Omron CX-Programmer project NewProject (CX-Programmer 9.61)

# PLC NewPLC1: CJ2M CPU35
I/O table (CPU CJ2M-CPU35): rack 0 slot 0 CJ1W-ID211; rack 0 slot 1 CJ1W-ID211; rack 0 slot 2 CJ1W-ID211; rack 0 slot 3 CJ1W-ID211; rack 0 slot 4 CJ1W-ID211; rack 0 slot 5 CJ1W-OD211; rack 0 slot 6 CJ1W-OD211; rack 0 slot 7 CJ1W-OD211; rack 0 slot 11 CJ2M-EIP21

## Global symbols (name address type ; comment)
0.00 BOOL  ; EMERGENCY STOP
0.01 BOOL  ; ALARM INVERTER 1
0.02 BOOL  ; ALARM INVERTER 2
0.03 BOOL  ; ALARM INVERTER 3
0.04 BOOL  ; ALARM INVERTER 4
0.05 BOOL  ; ALARM INVERTER 5
0.06 BOOL  ; ALARM INVERTER 6
0.07 BOOL  ; ALARM INVERTER 7
0.08 BOOL  ; ALARM INVERTER 8 FAULT
0.09 BOOL  ; ALARM INVERTER 9
0.10 BOOL  ; ALARM INVERTER 10
0.11 BOOL  ; PH1
0.12 BOOL  ; PH2
0.13 BOOL  ; PH3
0.14 BOOL  ; PH4
0.15 BOOL  ; PH5
100 CHANNEL  ; COUNTER MATERIAL M10
1000 CHANNEL  ; HOMEPOST VALUE
10.00 BOOL  ; IR MAN M1 FWD
10.01 BOOL  ; IR MAN M1 RVS
10.02 BOOL  ; IR MAN M2 FWD
10.03 BOOL  ; IR MAN M2 RVS
10.04 BOOL  ; IR MAN M3 FWD
10.05 BOOL  ; IR MAN M3 RVS
10.06 BOOL  ; IR MAN M4 FWD
10.07 BOOL  ; IR MAN M4 RVS
10.08 BOOL  ; IR MAN M5 FWD
10.09 BOOL  ; IR MAN M5 RVS
10.10 BOOL  ; IR MAN M6 FWD
10.11 BOOL  ; IR MAN M6 RVS
10.12 BOOL  ; IR MAN M7 FWD
10.13 BOOL  ; IR MAN M7 RVS
10.14 BOOL  ; IR MAN M8 FWD
10.15 BOOL  ; IR MAN M8 RVS
11.00 BOOL  ; IR MAN M9 FWD
11.01 BOOL  ; IR MAN M9 RVS
11.02 BOOL  ; IR MAN M10 FWD
11.03 BOOL  ; IR MAN M10 RVS
11.04 BOOL  ; IR MASTER ON
11.05 BOOL  ; MASTER OFF
11.06 BOOL  ; IR AUTO
11.07 BOOL  ; IR MANUAL
11.08 BOOL  ; IR MAN STP1 UP
11.09 BOOL  ; IR MAN STP1 DN
11.10 BOOL  ; IR MAN STP2 UP
11.11 BOOL  ; IR MAN STP2 DN
11.12 BOOL  ; IR MAN STP3 UP
11.13 BOOL  ; IR MAN STP3 DN
11.14 BOOL  ; IR MAN STP4 UP
11.15 BOOL  ; IR MAN STP4 DN
12.00 BOOL  ; IR MAN STP5 UP
12.01 BOOL  ; IR MAN STP5 DN
12.02 BOOL  ; IR MAN STP6 UP
12.03 BOOL  ; IR MAN STP6 DN
12.04 BOOL  ; IR MAN STP7 UP
12.05 BOOL  ; IR MAN STP7 DN
12.06 BOOL  ; IR MAN STP8 UP
12.07 BOOL  ; IR MAN STP8 DN
12.08 BOOL  ; IR MAN STP9 UP
12.09 BOOL  ; IR MAN STP9 DN
12.10 BOOL  ; IR MAN STP10 UP
12.11 BOOL  ; IR MAN STP10 DN
12.12 BOOL  ; IR MAN STP11 UP
12.13 BOOL  ; IR MAN STP11 DN
12.14 BOOL  ; IR MAN STP12 UP
12.15 BOOL  ; IR MAN STP12 DN
13.00 BOOL  ; IR MAN STP13 UP
13.01 BOOL  ; IR MAN STP13 DN
13.02 BOOL  ; IR MAN STP14 UP
13.03 BOOL  ; IR MAN STP14 DN
13.04 BOOL  ; IR HMI IN MOTOR ROLLER4 FWD
13.05 BOOL  ; IR HMI IN MOTOR ROLLER4 RVS
13.06 BOOL  ; IR HMI IN MOTOR ROLLER3 FWD
13.07 BOOL  ; IR HMI IN MOTOR ROLLER3 RVS
13.08 BOOL  ; IR HMI IN MOTOR ROLLER2 FWD
13.09 BOOL  ; IR HMI IN MOTOR ROLLER2 RVS
13.10 BOOL  ; IR HMI IN MOTOR ROLLER1 FWD
13.11 BOOL  ; IR HMI IN MOTOR ROLLER1 RVS
13.12 BOOL  ; START AUTO SEQUENCE
13.13 BOOL  ; FAULT MOTOR CONFIRM
13.14 BOOL  ; MAN PINLOCK UP ROT4
13.15 BOOL  ; MAN PINLOCK DOWN ROT4
14.00 BOOL  ; MAN PINLOCK UP ROT3
14.01 BOOL  ; MAN PINLOCK DOWN ROT3
14.02 BOOL  ; MAN PINLOCK UP ROT2
14.03 BOOL  ; MAN PINLOCK ROT2 DOWN
14.04 BOOL  ; MAN PINLOCK ROT1 UP
14.05 BOOL  ; MAN PINLOCK ROT1 DOWN
14.07 BOOL  ; FLAG DATA
14.08 BOOL  ; RECEIVE DATA BUFFER FULL FLAG
14.09 BOOL  ; IR PH23
14.10 BOOL  ; IR PH1
14.11 BOOL  ; IR PH2
14.12 BOOL  ; IR PH3
14.13 BOOL  ; IR PH4
14.14 BOOL  ; IR PH5
14.15 BOOL  ; IR PH6
15.00 BOOL  ; IR PH7
15.01 BOOL  ; IR PH8
15.02 BOOL  ; IR PH9
15.03 BOOL  ; IR PH10
15.04 BOOL  ; IR PH11
15.05 BOOL  ; IR PH12
15.06 BOOL  ; IR PH13
15.07 BOOL  ; IR PH14
15.08 BOOL  ; IR PH15
15.09 BOOL  ; IR PH16
15.10 BOOL  ; IR PH17
15.11 BOOL  ; IR PH18
15.12 BOOL  ; IR PH19
15.13 BOOL  ; IR PH20
15.14 BOOL  ; IR PH21
15.15 BOOL  ; IR PH22
16.00 BOOL  ; AUTO IN MATERIAL M10 FWD
16.01 BOOL  ; AUTO IN MATERIAL M9 FWD
16.02 BOOL  ; AUTO IN ROLLER1 FWD
16.03 BOOL  ; AUTO DOWN STP10
16.04 BOOL  ; CONFIRM ROT 1 STRAIGHT
16.05 BOOL  ; AUTO STP12 DOWN
16.06 BOOL  ; AUTO UP STP12
16.07 BOOL  ; AUTO STP11 DN
16.08 BOOL  ; AUTO UP STP11
16.09 BOOL  ; AUTO DOWN STP10 TURN
16.10 BOOL  ; AUTO MTR ROT1 TURN
16.11 BOOL  ; CONFIRM ROT 1 TURN
16.12 BOOL  ; AUTO OUT ROL1 FWD
16.13 BOOL  ; AUTO IN FWD M7
16.14 BOOL  ; AUTO STP10 UP
17.00 BOOL  ; AUTO STP10 UP TURN
17.01 BOOL  ; CONFIRM TRANFER OUT TURN ROT 1
17.02 BOOL  ; AUTO BACK STRAIGHT AFTER TRANFER TURN
17.03 BOOL  ; AUTO STP13 DOWN
17.04 BOOL  ; AUTO OUT MATERIAL M10 FWD
17.05 BOOL  ; AUTO UP STP13 AFTER OUT MATERIAL
17.06 BOOL  ; AUTO OUT MATERIAL M9 FWD
17.07 BOOL  ; AUTO OUT STP9 DOWN
17.08 BOOL  ; AUTO OUT M7 FWD
17.09 BOOL  ; AUTO UP STP9 AFTER TRANSFER
17.10 BOOL  ; AUTO IN DOWN STP8
17.11 BOOL  ; AUTO IN M ROLLER 2 FWD
17.12 BOOL  ; AUTO OUT M.ROLLER2 FWD
17.13 BOOL  ; AUTO MROT2 FWD
17.14 BOOL  ; AUTO MROT2 RVS
17.15 BOOL  ; AUTO PINLOCK2 UP
18.00 BOOL  ; AUTO PINLOCK2 DOWN
18.01 BOOL  ; AUTO STP8 UP
18.02 BOOL  ; AUTO STP8 DOWN
18.03 BOOL  ; AUTO STP7 UP
18.04 BOOL  ; AUTO STP7 DOWN
18.05 BOOL  ; CONFIRM TRANSFER SEGMEN 3
18.06 BOOL  ; AUTO STP14 DOWN
18.07 BOOL  ; AUTO IN M5 FWD
18.08 BOOL  ; AUTO STP6 DOWN
18.09 BOOL  ; AUTO OUT M5 FWD
18.10 BOOL  ; AUTO STP6 UP AFTER TRANFER
18.11 BOOL  ; AUTO IN M.ROLLER3 FWD
18.12 BOOL  ; AUTO OUT M.ROLLER3 FWD
18.13 BOOL  ; AUTO M.ROT3 FWD
18.14 BOOL  ; AUTO M.ROT3 RVS
18.15 BOOL  ; AUTO PINLOCK3 UP
19.00 BOOL  ; AUTO PINLOCK3 DOWN
19.01 BOOL  ; AUTO STP5 UP
19.02 BOOL  ; AUTO STP5 DOWN
19.03 BOOL  ; AUTO STP4 UP
19.04 BOOL  ; AUTO STP4 DOWN
19.05 BOOL  ; AUTO IN M3 FWD
19.06 BOOL  ; AUTO STP3 DOWN
19.07 BOOL  ; AUTO OUT M3 FWD
19.08 BOOL  ; AUTO STP3 UP
19.09 BOOL  ; AUTO STP14 UP
19.10 BOOL  ; IR RFID STRAIGHT CONFIRM
19.11 BOOL  ; IR RFID TURN CONFIRM 2
19.12 BOOL  ; AUTO IN M.ROLLER4 FWD
19.13 BOOL  ; AUTO OUT M.ROLLER4 FWD
19.14 BOOL  ; AUTO M.ROT4 FWD
19.15 BOOL  ; AUTO M.ROT4 RVS
1.00 BOOL  ; PH6
1.01 BOOL  ; PH7
1.02 BOOL  ; PH8
1.03 BOOL  ; PH9
1.04 BOOL  ; PH10
1.05 BOOL  ; PH11
1.06 BOOL  ; PH12
1.07 BOOL  ; PH13
1.08 BOOL  ; PH14
1.09 BOOL  ; PH15
1.10 BOOL  ; PH 16
1.11 BOOL  ; PH17
1.12 BOOL  ; PH18
1.13 BOOL  ; PH19
1.14 BOOL  ; PH20
1.15 BOOL  ; PH21
200 CHANNEL  ; LAST RFID DATA TO ROT1
20.00 BOOL  ; PINLOCK4 UP
20.01 BOOL  ; PINLOCK4 DOWN
20.02 BOOL  ; AUTO STP2 UP
20.03 BOOL  ; AUTO STP2 DOWN
20.04 BOOL  ; AUTO STP1 UP
20.05 BOOL  ; AUTO STP1 DOWN
20.06 BOOL  ; AUTO M1 FWD
20.07 BOOL  ; AUTO PINLOCK1 UP
20.08 BOOL  ; AUTO PINLOCK1 DOWN
20.09 BOOL  ; RESET HMI IN
20.10 BOOL  ; IR HMI MOTOR ROLLER5 FWD
20.11 BOOL  ; IR HMI MOTOR ROLLER5 RVS
20.12 BOOL  ; IR RFID 1 TURN CONFIRM
20.14 BOOL  ; IR RFID 2 CONFIRM TURN
21.00 BOOL  ; IR RFID 3 CONFIRM TURN
21.02 BOOL  ; IR RFID 4 CONFIRM TURN
21.03 BOOL  ; IR RFID 4 CONFIRM STRAIGHT
21.04 BOOL  ; RFID ROT1 ON
21.05 BOOL  ; RFID ROT3 ON
21.06 BOOL  ; IR RFID 5 CONFIRM STRAIGHT
21.08 BOOL  ; IR MAN PINLOCK ROT4 UP
21.09 BOOL  ; IR MAN PINLOCK ROT4 DN
21.10 BOOL  ; IR MAN PIN LOCK ROT3 UP
21.11 BOOL  ; IR MAN PIN LOCK ROT3 DN
21.12 BOOL  ; IR MAN PIN LOCK ROT2 UP
21.13 BOOL  ; IR MAN PIN LOCK ROT2 DN
21.14 BOOL  ; IR MAN PIN LOCK ROT1 UP
21.15 BOOL  ; IR MAN PIN LOCK ROT1 DN
22.00 BOOL  ; HALF RADIUS IN
22.01 BOOL  ; AUTO IN ROLLER5 FWD
22.02 BOOL  ; AUTO OUT ROLLER5 FWD
23.00 BOOL  ; IR ROLLER IN ROT1 ON
23.01 BOOL  ; IR ROLLER IN ROT2 ON
23.02 BOOL  ; IR ROLLER IN ROT3 ON
23.03 BOOL  ; IR ROLLER IN ROT4 ON
28.00 BOOL  ; EMERGENCY PUSHED
29.00 BOOL  ; HMI OUT MASTER ON
29.01 BOOL  ; HMI OUT AUTO/MAN INDI
29.02 BOOL  ; HMI OUT INDI AIR ON
29.04 BOOL  ; HMI LIST MASTER OFF
29.05 BOOL  ; HMI LIST AIR PRESSURE OFF
29.06 BOOL  ; HMI LIST INVERTER 1 FAULT
29.07 BOOL  ; HMI LIST INVERTER 2 FAULT
29.08 BOOL  ; HMI LIST INVERTER 3 FAULT
29.09 BOOL  ; HMI INVERTER 4 FAULT
29.10 BOOL  ; HMI INVERTER 5 FAULT
29.11 BOOL  ; HMI INVERTER 6 FAULT
29.12 BOOL  ; HMI LIST INVERTER 7 FAULT
29.13 BOOL  ; HMI LIST INVERTER 8 FAULT
29.14 BOOL  ; HMI LIST INVERTER 9 FAULT
29.15 BOOL  ; HMI LIST INVERTER 10 FAULT
2.00 BOOL  ; PH22
2.01 BOOL  ; RSDN STP13
2.02 BOOL  ; RSUP STP13
2.03 BOOL  ; RSDN STP12
2.04 BOOL  ; RSUP STP12
2.05 BOOL  ; RSDN STP11
2.06 BOOL  ; RSUP STP11
2.07 BOOL  ; RSDN STP10
2.08 BOOL  ; RSUP STP10
2.09 BOOL  ; RSDN STP9
2.10 BOOL  ; RSUP STP9
2.11 BOOL  ; RSDN STP8
2.12 BOOL  ; RSUP STP8
2.13 BOOL  ; RSDN STP7
2.14 BOOL  ; RSUP STP7
2.15 BOOL  ; RSUP STP6
30.00 BOOL  ; HMI IN M1 FWD
30.01 BOOL  ; HMI IN M1 RVS
30.02 BOOL  ; HMI IN M2 FWD
30.03 BOOL  ; HMI IN M2 RVS
30.04 BOOL  ; HMI IN M3 FWD
30.05 BOOL  ; HMI IN M3 RVS
30.06 BOOL  ; HMI IN M4 FWD
30.07 BOOL  ; HMI IN M4 RVS
30.08 BOOL  ; HMI IN M5 FWD
30.09 BOOL  ; HMI IN M5 RVS
30.10 BOOL  ; HMI IN M6 FWD
30.11 BOOL  ; HMI IN M6 RVS
30.12 BOOL  ; HMI IN M7 FWD
30.13 BOOL  ; HMI IN M7 RVS
30.14 BOOL  ; HMI IN M8 FWD
30.15 BOOL  ; HMI IN M8 RVS
31.00 BOOL  ; HMI IN M9 FWD
31.01 BOOL  ; HMI IN M9 RVS
31.02 BOOL  ; HMI IN M10 FWD
31.03 BOOL  ; HMI IN M10 RVS
31.04 BOOL  ; INDI HMI M1 FWD
31.05 BOOL  ; INDI HMI M1 RVS
31.06 BOOL  ; INDI HMI ROT 4 TURN
31.07 BOOL  ; INDI HMI ROT 4 STRAIGHT
31.08 BOOL  ; INDI HMI M3 FWD
31.09 BOOL  ; INDI HMI M3 RVS
31.10 BOOL  ; INDI HMI ROT 3 TURN
31.11 BOOL  ; INDI HMI ROT 3 STRAIGHT
31.12 BOOL  ; INDI HMI M5 FWD
31.13 BOOL  ; INDI HMI M5 RVS
31.14 BOOL  ; INDI HMI ROT 2 TURN
31.15 BOOL  ; INDI HMI ROT 2 STRAIGHT
3201.00 BOOL  ; SW AUT/MAN
3201.01 BOOL  ; PB START
3201.02 BOOL  ; ALARM ROLLER 4
3201.03 BOOL  ; PB RESET
3201.04 BOOL  ; ALARM ROLLER 3
3201.05 BOOL  ; PB EXECUTE
3201.06 BOOL  ; ALARM ROLLER 2
3201.07 BOOL  ; MASTER ON
3201.08 BOOL  ; AIR PRESSURE SWITCH
3201.09 BOOL  ; ALARM ROLLER 1
3201.10 BOOL  ; ANTENA RFID OFF
3201.11 BOOL  ; ALARM ROLLER HALF RADIUS
3201.12 BOOL  ; INTERLOCK ROT4
3201.13 BOOL  ; INTERLOCK ROT3
3201.14 BOOL  ; INTERLOCK ROT2
3201.15 BOOL  ; INTERLOCK ROT1
3202.03 BOOL  ; RECIEVE DATA BUFFER FULL FLAG
3203 CHANNEL  ; DATA IN
3205.01 BOOL  ; FLAG DATA
3210 CHANNEL  ; DATA NO ANTENA
3216 CHANNEL  ; FIRST DATA IN HMI
32.00 BOOL  ; INDI HMI M7 FWD
32.01 BOOL  ; INDI HMI M7 RVS
32.02 BOOL  ; INDI HMI ROT 1 TURN
32.03 BOOL  ; INDI HMI ROT 1 STRAIGHT
32.04 BOOL  ; INDI HMI M9 FWD
32.05 BOOL  ; INDI HMI M9 RVS
32.06 BOOL  ; INDI HMI M10 FWD
32.07 BOOL  ; INDI HMI M10 RVS
32.08 BOOL  ; HMI IN STP1 UP
32.09 BOOL  ; HMI IN STP1 DN
32.10 BOOL  ; HMI IN STP2 UP
32.11 BOOL  ; HMI IN STP2 DN
32.12 BOOL  ; HMI IN STP3 UP
32.13 BOOL  ; HMI IN STP3 DN
32.14 BOOL  ; HMI IN STP4 UP
32.15 BOOL  ; HMI IN STP4 DN
3300.00 BOOL  ; TOWER LAMP GREEN
3300.01 BOOL  ; TOWER LAMP YELLOW
3300.02 BOOL  ; TOWER LAMP RED
3300.03 BOOL  ; BUZZER FAULT CONFIRM ON
3300.04 BOOL  ; OUT STP1 DN
3300.05 BOOL  ; OUT STP1 UP
3300.06 BOOL  ; OUT STP2 DN
3300.07 BOOL  ; OUT STP2 UP
3300.08 BOOL  ; OUT STP3 DN
3300.09 BOOL  ; OUT STP3 UP
3300.10 BOOL  ; OUT STP4 DN
3300.11 BOOL  ; OUT STP4 UP
3300.12 BOOL  ; OUT STP5 DN
3300.13 BOOL  ; OUT STP5 UP
3300.14 BOOL  ; OUT STP6 DN
3300.15 BOOL  ; OUT STP6 UP
3301.00 BOOL  ; OUT STP7 DN
3301.01 BOOL  ; OUT STP7 UP
3301.02 BOOL  ; OUT STP8 DN
3301.03 BOOL  ; OUT STP8 UP
3301.04 BOOL  ; OUT STP9 DN
3301.05 BOOL  ; OUT STP9 UP
3301.06 BOOL  ; OUT STP10 DN
3301.07 BOOL  ; OUT STP10 UP
3301.08 BOOL  ; OUT STP11 DN
3301.09 BOOL  ; OUT STP11 UP
3301.10 BOOL  ; OUT STP12 DN
3301.11 BOOL  ; OUT STP12 UP
3301.12 BOOL  ; OUT STP13 DN
3301.13 BOOL  ; OUT STP13 UP
3301.14 BOOL  ; OUT STP14 DN
3301.15 BOOL  ; OUT STP14 UP
3302.00 BOOL  ; OUT PINLOCK ROT4 UP
3302.01 BOOL  ; OUT PINLOCK ROT4 DN
3302.02 BOOL  ; OUT PINLOCK ROT1 DN
3302.03 BOOL  ; OUT PINLOCK ROT1 UP
3302.04 BOOL  ; OUT PINLOCK ROT2 DN
3302.05 BOOL  ; OUT PINLOCK ROT2 UP
3302.06 BOOL  ; OUT PINLOCK ROT3 DN
3302.07 BOOL  ; OUT PINLOCK ROT3 UP
3302.09 BOOL  ; OUT M.ROLLER5 FWD
3302.10 BOOL  ; OUT M ROLLER5 RVS
3302.12 BOOL  ; RESET ALL ROLLER
3303 CHANNEL  ; OUT DATA
33.00 BOOL  ; HMI IN STP5 UP
33.01 BOOL  ; HMI IN STP5 DN
33.02 BOOL  ; HMI IN STP6 UP
33.03 BOOL  ; HMI IN STP6 DN
33.04 BOOL  ; HMI IN STP7 UP
33.05 BOOL  ; HMI IN STP7 DN
33.06 BOOL  ; HMI IN STP8 UP
33.07 BOOL  ; HMI IN STP8 DN
33.08 BOOL  ; HMI IN STP9 UP
33.09 BOOL  ; HMI IN STP9 DN
33.10 BOOL  ; HMI IN STP10 UP
33.11 BOOL  ; HMI IN STP10 DN
33.12 BOOL  ; HMI IN STP11 UP
33.13 BOOL  ; HMI IN STP11 DN
33.14 BOOL  ; HMI IN STP12 UP
33.15 BOOL  ; HMI IN STP12 DN
34.00 BOOL  ; HMI IN STP13 UP
34.01 BOOL  ; HMI IN STP13 DN
34.02 BOOL  ; HMI IN STP14 UP
34.03 BOOL  ; HMI IN STP14 DN
34.04 BOOL  ; HMI INDI RSUP STP1
34.05 BOOL  ; HMI INDI RSDN STP1
34.06 BOOL  ; HMI INDI RSUP STP2
34.07 BOOL  ; HMI INDI RSDN STP2
34.08 BOOL  ; HMI INDI RSUP STP3
34.09 BOOL  ; HMI INDI RSDN STP3
34.10 BOOL  ; HMI INDI RSUP STP4
34.11 BOOL  ; HMI INDI RSDN STP4
34.12 BOOL  ; HMI INDI RSUP STP5
34.13 BOOL  ; HMI INDI RSDN STP5
34.14 BOOL  ; HMI INDI RSUP STP6
34.15 BOOL  ; HMI INDI RSDN STP6
35.00 BOOL  ; HMI INDI RSUP STP7
35.01 BOOL  ; HMI INDI RSDN STP7
35.02 BOOL  ; HMI INDI RSUP STP8
35.03 BOOL  ; HMI INDI RSDN STP8
35.04 BOOL  ; HMI INDI RSUP STP9
35.05 BOOL  ; HMI INDI RSDN STP9
35.06 BOOL  ; HMI INDI RSUP STP10
35.07 BOOL  ; HMI INDI RSDN STP10
35.08 BOOL  ; HMI INDI RSUP STP11
35.09 BOOL  ; HMI INDI RSDN STP11
35.10 BOOL  ; HMI INDI RSUP STP12
35.11 BOOL  ; HMI INDI RSDN STP12
35.12 BOOL  ; HMI INDI RSUP STP13
35.13 BOOL  ; HMI INDI RSDN STP13
35.14 BOOL  ; HMI IN MOTOR ROLLER4 FWD
35.15 BOOL  ; HMI IN MOTOR ROLLER4 RVS
36.00 BOOL  ; HMI IN MOTOR ROLLER3 FWD
36.01 BOOL  ; HMI IN MOTOR ROLLER3 RVS
36.02 BOOL  ; HMI IN MOTOR ROLLER2 FWD
36.03 BOOL  ; HMI IN MOTOR ROLLER2 RVS
36.04 BOOL  ; HMI IN MOTOR ROLLER1 FWD
36.05 BOOL  ; HMI IN MOTOR ROLLER1 RVS
36.06 BOOL  ; HMI INDI MOTOR ROLLER4 FWD
36.07 BOOL  ; HMI INDI MOTOR ROLLER4 RVS
36.08 BOOL  ; HMI INDI MOTOR ROLLER3 FWD
36.09 BOOL  ; HMI INI MOTOR ROLLER3 RVS
36.10 BOOL  ; HMI INDI MOTOR ROLLER2 FWD
36.11 BOOL  ; HMI INDI MOTOR ROLLER2 RVS
36.12 BOOL  ; HMI INDI MOTOR ROLLER1 FWD
36.13 BOOL  ; HMI INDI MOTOR ROLLER1 RVS
36.14 BOOL  ; HMI IN PINLOCK ROT4 UP
36.15 BOOL  ; HMI IN PINLOCK ROT4 DN
37.00 BOOL  ; HMI IN PINLOCK ROT3 UP
37.01 BOOL  ; HMI IN PINLOCK ROT3 DN
37.02 BOOL  ; HMI IN PINLOCK ROT2 UP
37.03 BOOL  ; HMI IN PIN LOCK ROT2 DN
37.04 BOOL  ; HMI IN PINLOCK ROT1 UP
37.05 BOOL  ; HMI IIN PIN LOCK ROT1 DN
37.06 BOOL  ; RFID RECIEVE DATA
37.08 BOOL  ; RFID 1 STRAIGHT
37.09 BOOL  ; RFID 1 TURN
37.10 BOOL  ; HMI INDI RSUP PINLOCK ROT1
37.11 BOOL  ; HMI INDI RSDN PINLOCK ROT1
37.12 BOOL  ; HMI INDI RSUP PINLOCK ROT2
37.13 BOOL  ; HMI INDI RSUP PINLOCK ROT2
37.14 BOOL  ; HMI INDI RSUP PINLOCK ROT3
37.15 BOOL  ; HMI INDI RSDN PINLOCK ROT3
38.00 BOOL  ; HMI INDI RSUP PINLOCK ROT4
38.01 BOOL  ; HMI INDI RSDN PINLOCK ROT4
38.02 BOOL  ; HMI INDI RSUP STP14
38.03 BOOL  ; HMI INDI RSDN STP14
38.04 BOOL  ; RFID STRAIGHT CONFIRM 2
38.05 BOOL  ; RFID TURN CONFIRM 2
38.06 BOOL  ; RFID STRAIGHT CONFIRM 3
38.07 BOOL  ; RFID TURN CONFIRM 3
38.08 BOOL  ; RFID STRAIGHT CONFIRM 4
38.09 BOOL  ; RFID TURN CONFIRM 4
38.10 BOOL  ; ENABLE READER
38.10 BOOL  ; ENABLE RFID
38.14 BOOL  ; PB SAVE 1
38.15 BOOL  ; PB SAVE 2
39.00 BOOL  ; HMI PB SAVE 3
39.01 BOOL  ; HMI PB SAVE 4
39.02 BOOL  ; PB HMI CLEAR MEMORY 1
39.03 BOOL  ; PB HMI HOME POST
39.04 BOOL  ; PB HMI CLEAR MEMORY 2
39.05 BOOL  ; HMI IND HOME POST
39.06 BOOL  ; PB HMI CLEAR MEMORY 3
39.07 BOOL  ; HMI PB STRAIGHT 3
39.08 BOOL  ; PB HMI CLEAR MEMORY 4
39.09 BOOL  ; HMI PB STRAIGHT 4
39.10 BOOL  ; PB HMI PREV
39.11 BOOL  ; PB HMI NEXT
39.12 BOOL  ; PB HMI PREV 2
39.13 BOOL  ; PB HMI NEXT 2
39.14 BOOL  ; PB HMI PREV 3
39.15 BOOL  ; PB HMI NEXT 3
3.00 BOOL  ; RSDN STP6
3.01 BOOL  ; RSUP STP5
3.02 BOOL  ; RSDN STP5
3.03 BOOL  ; RSUP STP4
3.04 BOOL  ; RSDN STP4
3.05 BOOL  ; RSUP STP3
3.06 BOOL  ; RSDN STP3
3.07 BOOL  ; RSUP STP2
3.08 BOOL  ; RSDN STP2
3.09 BOOL  ; RSUP STP1
3.10 BOOL  ; RSDN STP1
3.11 BOOL  ; RSUP STP14
3.12 BOOL  ; RSDN STP14
3.14 BOOL  ; PH 23
40.00 BOOL  ; PB HMI PREV 4
40.01 BOOL  ; PB HMI NEXT 4
40.02 BOOL  ; IR CAN PUSH PB SAVE1 HMI
40.03 BOOL  ; HMI IN MOTOR ROLLER 5 FWD
40.04 BOOL  ; HMI IN MOTOR ROLLER5 RVS
40.05 BOOL  ; HMI IN M. ROLLER5 FWD
40.06 BOOL  ; HMI INDI M.ROLLER5 RVS
40.07 BOOL  ; DONE STRAIGHT ROT 1
40.08 BOOL  ; DONE TURN ROT 1
40.09 BOOL  ; DONE STRAIGHT ROT 2
40.10 BOOL  ; DONE TURN ROT 2
40.11 BOOL  ; DONE STRAIGHT ROT 3
40.12 BOOL  ; DONE TURN ROT 3
40.13 BOOL  ; DONE STRAIGHT ROT 4
40.14 BOOL  ; DONE TURN ROT 4
40.15 BOOL  ; CONFIRM TURN 2
41.00 BOOL  ; PH OUT AFTER ROT1
41.01 BOOL  ; MOTOR CONV AFTER ROT1
41.02 BOOL  ; PH OUT AFTER ROT2
41.03 BOOL  ; MOTOR CONV AFTER ROT2
41.04 BOOL  ; PH OUT AFTER ROT3
41.05 BOOL  ; MOTOR CONV AFTER ROT3
41.06 BOOL  ; HMI PB SAVE 5
41.07 BOOL  ; PB HMI CLEAR MEMORY 5
41.08 BOOL  ; PB HMI PREV 5
41.09 BOOL  ; PB HMI NEXT 5
42.00 BOOL  ; HOMEPOST DONE 1
42.01 BOOL  ; HOMEPOST DONE 2
42.02 BOOL  ; HOMEPOST DONE 3
42.03 BOOL  ; HOMEPOST DONE 4
42.04 BOOL  ; HOMEPOST DONE ALL
42.05 BOOL  ; READY AUTO
42.06 BOOL  ; AFTER FIRST HOMEPOST
43.00 BOOL  ; TIMER PH6
43.01 BOOL  ; TIMER PH10
43.02 BOOL  ; TIMER PH14
43.03 BOOL  ; TIMER PH18
45.02 BOOL  ; YELLOW LAMP FLASH
45.03 BOOL  ; YELLOW LAMP LIT
45.04 BOOL  ; FLASHING IND
45.05 BOOL  ; HMI LIST ROLLER 4 FAULT
45.06 BOOL  ; HMI LIST ROLLER 3 FAULT
45.07 BOOL  ; HMI LIST ROLLER 2 FAULT
45.08 BOOL  ; HMI LIST ROLLER 1 FAULT
45.09 BOOL  ; HMI LIST ROLLER HALF RADIUS FAULT
45.10 BOOL  ; DELAY AWAITING M10 IN
45.11 BOOL  ; DATA IN INC PH1
45.12 BOOL  ; DATA IN DEC PHS 2
45.13 BOOL  ; REFRESH RFID HMI
45.14 BOOL  ; IND RFID DETECT HMI
45.15 BOOL  ; IR NUMBER RFID SWAP
46.00 BOOL  ; RFID 1 DATA REDUDANCY ALARM
46.01 BOOL  ; RFID 2 DATA REDUDANCY ALARM
46.02 BOOL  ; RFID 3 DATA REDUDANCY ALARM
46.03 BOOL  ; RFID 4 DATA REDUDANCY ALARM
46.04 BOOL  ; REDUDANCY RFID 1 ACCEPTED
46.05 BOOL  ; REDUDANCY RFID 2 ACCEPTED
46.06 BOOL  ; REDUDANCY RFID 3 ACCEPTED
46.07 BOOL  ; REDUDANCY RFID 4 ACCEPTED
46.08 BOOL  ; HMI RFID DATA REDUDANCY
46.09 BOOL  ; HMI REDUDANCY RFID ACCEPTED
46.10 BOOL  ; REDUDANCY RFID 5 ACCEPTED
46.11 BOOL  ; RFID 5 DATA REDUDANCY ALARM
46.12 BOOL  ; DONE ACQUIRE RFID NUMBER AUTO
46.13 BOOL  ; DONE ACQUIRE RFID NUMBER MANUAL
47.00 BOOL  ; TRANSFER FROM CONV 10
47.01 BOOL  ; TRANSFER FROM CONV 9
47.02 BOOL  ; TRANSFER FROM CONV 7
47.03 BOOL  ; TRANSFER FROM CONV 5
47.04 BOOL  ; TRANSFER FROM CONV 3
47.05 BOOL  ; AWAITING STP14 DOWN
48.00 BOOL  ; FAULT INV 1
48.01 BOOL  ; FAULT INV 2
48.02 BOOL  ; FAULT INV 3
48.03 BOOL  ; FAULT INV 4
48.04 BOOL  ; FAULT INV 5
48.05 BOOL  ; FAULT INV 6
48.06 BOOL  ; FAULT INV 7
48.07 BOOL  ; FAULT INV 8
48.08 BOOL  ; FAULT INV 9
48.09 BOOL  ; FAULT INV 10
48.10 BOOL  ; FAULT ROLLER 4
48.11 BOOL  ; FAULT ROLLER 3
48.12 BOOL  ; FAULT ROLLER 2
48.13 BOOL  ; FAULT ROLLER 1
48.14 BOOL  ; FAULT ROLLER HALF RADIUS
4.00 BOOL  ; LS STRAIGHT ROT1
4.01 BOOL  ; LS TURN ROT1
4.02 BOOL  ; LS STRAIGTH ROT2
4.03 BOOL  ; LS TURN ROT2
4.04 BOOL  ; LS STRAIGHT ROT3
4.05 BOOL  ; LS.TURN ROT3
4.06 BOOL  ; LS STRAIGHT ROT4
4.07 BOOL  ; LS TURN ROT4
4.08 BOOL  ; RSUP PINLOCK ROT1
4.09 BOOL  ; RSDN PINLOCK ROT1
4.10 BOOL  ; RSUP PINLOCK ROT2
4.11 BOOL  ; RSDN PINLOCK ROT2
4.12 BOOL  ; RSUP PINLOCK ROT3
4.13 BOOL  ; RSDN PINLOCK ROT3
4.14 BOOL  ; RSUP PINLOCK ROT4
4.15 BOOL  ; RSDN PINLOCK ROT4
50.00 BOOL  ; CONFIRM STRAIGHT 2
50.01 BOOL  ; CONFIRM TURN 3
50.02 BOOL  ; CONFIRM STRAIGHT 3
50.03 BOOL  ; IR CAN PUSH PB SAVE 2 HMI
50.04 BOOL  ; IR CAN PUSH PB SAVE 3 HMI
50.05 BOOL  ; IR CAN PUSH SAVE 4 HMI
50.06 BOOL  ; CONFIRM TURN 4
50.07 BOOL  ; IR ENABLE CAN ON
5.00 BOOL  ; OUT M9 FWD
5.01 BOOL  ; OUT M9 RVS
5.02 BOOL  ; OUT M10 FWD
5.03 BOOL  ; OUT M10 RVS
5.04 BOOL  ; OUT M3 FWD
5.05 BOOL  ; OUT M3 RVS
5.06 BOOL  ; OUT M4 FWD
5.07 BOOL  ; OUT M4 RVS
5.08 BOOL  ; OUT M5 FWD
5.09 BOOL  ; OUT M5 RVS
5.10 BOOL  ; OUT M6 FWD
5.11 BOOL  ; OUT M6 RVS
5.12 BOOL  ; OUT M2 FWD
5.13 BOOL  ; OUT M2 RVS
5.14 BOOL  ; OUT M8 FWD
5.15 BOOL  ; OUT M8 RVS
60.00 BOOL  ; ALARM RFID NOT DETECT
60.01 BOOL  ; FAULT
60.04 BOOL  ; ALARM RFID 1 NOT DETECT
60.05 BOOL  ; ALARM RFID 2 NOT DETECT
60.06 BOOL  ; ALARM RFID 3 NOT DETECT
60.07 BOOL  ; ALARM RFID 4 NOT DETECT
60.08 BOOL  ; ALARM RFID NOT DETECT
60.09 BOOL  ; RFID OFF
60.10 BOOL  ; ALARM RFID 5 NOT DETECT
60.11 BOOL  ; HMI PREV BY PASS MATERIAL
60.12 BOOL  ; HMI NEXT BY PASS MATERIAL
6.00 BOOL  ; RSET INVERTER 1
6.01 BOOL  ; RESET INVERTER 2
6.02 BOOL  ; OUT MOTOR ROLLER4 FWD
6.03 BOOL  ; RESET INVERTER 3
6.04 BOOL  ; RESET INVERTER 4
6.05 BOOL  ; RESET INVERTER 5
6.06 BOOL  ; RESET INVERTER 6
6.07 BOOL  ; RESET INVERTER 7
6.08 BOOL  ; RESET INVERTER 8
6.09 BOOL  ; RESET INVERTER 9
6.10 BOOL  ; RESET INVERTER 10
6.11 BOOL  ; OUT MOTOR ROLLER4 RVS
6.12 BOOL  ; OUT MOTOR ROLLER3 FWD
6.13 BOOL  ; OUT MOTOR ROLLER3 RVS
6.14 BOOL  ; OUT MOTOR ROLLER2 FWD
6.15 BOOL  ; OUT MOTOR ROLLER2 RVS
70.00 BOOL  ; INTERLOCK HALF RADIUS
78.00 BOOL  ; HOMEPOST CONFIRM
7.00 BOOL  ; KONTAKTOR M9
7.01 BOOL  ; KONTAKTOR M10
7.02 BOOL  ; KONTAKTOR M3
7.03 BOOL  ; KONTAKTOR M4
7.04 BOOL  ; KONTAKTOR M5
7.05 BOOL  ; KONTAKTOR M6
7.06 BOOL  ; KONTAKTOR M2
7.07 BOOL  ; KONTAKTOR M8
7.08 BOOL  ; KONTAKTOR M1
7.09 BOOL  ; KONTAKTOR M7
7.10 BOOL  ; OUT M1 FWD
7.11 BOOL  ; OUT M1 RVS
7.12 BOOL  ; OUT M7 FWD
7.13 BOOL  ; OUT M7 RVS
7.14 BOOL  ; OUT MOTOR ROLLER1 FWD
7.15 BOOL  ; OUT MOTOR ROLLER1 RVS
80.00 BOOL  ; HOMEPOST STP1 UP
80.01 BOOL  ; HOMEPOST STP2 UP
80.02 BOOL  ; HOMEPOST STP3 UP
80.03 BOOL  ; HOMEPOST STP4 UP
80.04 BOOL  ; HOMEPOST STP5 UP
80.05 BOOL  ; HOMEPOST STP6 UP
80.06 BOOL  ; HOMEPOST STP7 UP
80.07 BOOL  ; HOMEPOST STP8 UP
80.08 BOOL  ; HOMEPOST STP9 UP
80.09 BOOL  ; HOMEPOST STP10 UP
80.10 BOOL  ; HOMEPOST STP11 UP
80.11 BOOL  ; HOMEPOST STP12 UP
80.12 BOOL  ; HOMEPOST STP13 UP
80.13 BOOL  ; HOMEPOST STP14 UP
80.14 BOOL  ; HOMEPOST ROT4 STRAIGHT
80.15 BOOL  ; HOMEPOST ROT3 STRAIGHT
81.00 BOOL  ; MATERIAL WAIT ON ROT 1
81.02 BOOL  ; SET CONFIRM STRAIGHT ROT 2
81.04 BOOL  ; SET CONFIRM STRAIGHT ORT 4
81.08 BOOL  ; MATERIAL WAIT ON ROT 2
81.09 BOOL  ; MATERIAL WAIT ON ROT 3
81.10 BOOL  ; SET CONFIRM TURN ROT 1
81.11 BOOL  ; SET CONFIRM STRAIGHT ROT 1
81.13 BOOL  ; IR MATERIAL WAIT BEFORE CONV 9
81.14 BOOL  ; CONFIRM STRAIGHT ROT 3
81.15 BOOL  ; MATERIAL CAN TRANFER TO AREA ROTARY
82.00 BOOL  ; STP 12 FORCE DOWN
82.01 BOOL  ; TURN ROT 1
82.02 BOOL  ; TURN ROT 2
82.03 BOOL  ; TURN ROT 3
82.04 BOOL  ; TURN ROT 4
82.05 BOOL  ; STRAIGHT ROT 4
82.06 BOOL  ; IR RFID 5 CONFIRM BUFFER CONV
82.07 BOOL  ; IR RFID 5 CONFIRM STRAIGHT
82.08 BOOL  ; RFID 5 DATA REDUDANCY ALARM
90.00 BOOL  ; HOMEPOST ROT2 STRAIGHT
90.01 BOOL  ; HOMEPOST ROT1 STRAIGHT
90.02 BOOL  ; PB HMI RVS ALL
90.03 BOOL  ; ALL MOTOR REVERSE
90.04 BOOL  ; ALL STOPPER DOWN
C0000 BOOL  ; COUNT 1
D0 CHANNEL  ; TEACHING RFID NO.1
D10 CHANNEL  ; TEACHING RFID NO 2
D1000 CHANNEL  ; MEMORY 1
D10000 CHANNEL  ; MEMORY 1
D10002 CHANNEL  ; MEMORY 2
D10004 CHANNEL  ; MEMORY 3
D10006 CHANNEL  ; MEMORY 4
D10008 CHANNEL  ; MEMORY 5
D10010 CHANNEL  ; MEMORY 6
D10012 CHANNEL  ; MEMORY 7
D10014 CHANNEL  ; MEMORY 8
D10016 CHANNEL  ; MEMORY 9
D10018 CHANNEL  ; MEMORY 10
D1002 CHANNEL  ; MEMORY 2
D10020 CHANNEL  ; MEMORY 11
D10022 CHANNEL  ; MEMORY 12
D10024 CHANNEL  ; MEMORY 13
D10026 CHANNEL  ; MEMORY 14
D10028 CHANNEL  ; MEMORY 15
D10030 CHANNEL  ; MEMORY 16
D10032 CHANNEL  ; MEMORY 17
D10034 CHANNEL  ; MEMORY 18
D10036 CHANNEL  ; MEMORY 19
D10038 CHANNEL  ; MEMORY 20
D1004 CHANNEL  ; MEMORY 3
D10040 CHANNEL  ; MEMORY 21
D10042 CHANNEL  ; MEMORY 22
D10044 CHANNEL  ; MEMORY 23
D10046 CHANNEL  ; MEMORY 24
D10048 CHANNEL  ; MEMORY 25
D10050 CHANNEL  ; MEMORY 26
D10052 CHANNEL  ; MEMORY 27
D10054 CHANNEL  ; MEMORY 28
D10056 CHANNEL  ; MEMORY 29
D10058 CHANNEL  ; MEMORY 30
D1006 CHANNEL  ; MEMORY 4
D10060 CHANNEL  ; MEMORY 31
D10062 CHANNEL  ; MEMORY 32
D10064 CHANNEL  ; MEMORY 33
D10066 CHANNEL  ; MEMORY 34
D10068 CHANNEL  ; MEMORY 35
D10070 CHANNEL  ; MEMORY 36
D10072 CHANNEL  ; MEMORY 37
D10074 CHANNEL  ; MEMORY 38
D10076 CHANNEL  ; MEMORY 39
D10078 CHANNEL  ; MEMORY 40
D1008 CHANNEL  ; MEMORY 5
D10080 CHANNEL  ; MEMORY 41
D10082 CHANNEL  ; MEMORY 42
D10084 CHANNEL  ; MEMORY 43
D10086 CHANNEL  ; MEMORY 44
D10088 CHANNEL  ; MEMORY 45
D10090 CHANNEL  ; MEMORY 46
D10092 CHANNEL  ; MEMORY 47
D10094 CHANNEL  ; MEMORY 48
D10096 CHANNEL  ; MEMORY 49
D10098 CHANNEL  ; MEMORY 50
D1010 CHANNEL  ; MEMORY 6
D1012 CHANNEL  ; MEMORY 7
D1014 CHANNEL  ; MEMORY 8
D1016 CHANNEL  ; MEMORY 9
D1018 CHANNEL  ; MEMORY 10
D1020 CHANNEL  ; MEMORY 11
D1022 CHANNEL  ; MEMORY 12
D1024 CHANNEL  ; MEMORY 13
D1026 CHANNEL  ; MEMORY 14
D1028 CHANNEL  ; MEMORY 15
D1030 CHANNEL  ; MEMORY 16
D1032 CHANNEL  ; MEMORY 17
D1034 CHANNEL  ; MEMORY 18
D1036 CHANNEL  ; MEMORY 19
D1038 CHANNEL  ; MEMORY 20
D1040 CHANNEL  ; MEMORY 21
D1042 CHANNEL  ; MEMORY 22
D1044 CHANNEL  ; MEMORY 23
D1046 CHANNEL  ; MEMORY 24
D1048 CHANNEL  ; MEMORY 25
D1050 CHANNEL  ; MEMORY 26
D10500 CHANNEL  ; HMI MONIT DEST
D1052 CHANNEL  ; MEMORY 27
D1054 CHANNEL  ; MEMORY 28
D1056 CHANNEL  ; MEMORY 29
D1058 CHANNEL  ; MEMORY 30
D1060 CHANNEL  ; MEMORY 31
D1062 CHANNEL  ; MEMORY 32
D1064 CHANNEL  ; MEMORY 33
D1066 CHANNEL  ; MEMORY 34
D1068 CHANNEL  ; MEMORY 35
D1070 CHANNEL  ; MEMORY 36
D1072 CHANNEL  ; MEMORY 37
D1074 CHANNEL  ; MEMORY 38
D1076 CHANNEL  ; MEMORY 39
D1078 CHANNEL  ; MEMORY 40
D1080 CHANNEL  ; MEMORY 41
D1082 CHANNEL  ; MEMORY 42
D1084 CHANNEL  ; MEMORY 43
D1086 CHANNEL  ; MEMORY 44
D1088 CHANNEL  ; MEMORY 45
D1090 CHANNEL  ; MEMORY 46
D1092 CHANNEL  ; MEMORY 47
D1094 CHANNEL  ; MEMORY 48
D1096 CHANNEL  ; MEMORY 49
D1098 CHANNEL  ; MEMORY 50
D140 CHANNEL  ; DISPLAY TEACH RFID 3 HMI
D20 CHANNEL  ; TEACH RFID 3
D200 CHANNEL  ; NO. READER 2
D2000 CHANNEL  ; MEMORY 1
D2002 CHANNEL  ; MEMORY 2
D2004 CHANNEL  ; MEMORY 3
D2006 CHANNEL  ; MEMORY 4
D2008 CHANNEL  ; MEMORY 5
D2010 CHANNEL  ; MEMORY 6
D2012 CHANNEL  ; MEMORY 7
D2014 CHANNEL  ; MEMORY 8
D2016 CHANNEL  ; MEMORY 9
D2018 CHANNEL  ; MEMORY 10
D2020 CHANNEL  ; MEMORY 11
D2022 CHANNEL  ; MEMORY 12
D2024 CHANNEL  ; MEMORY 13
D2026 CHANNEL  ; MEMORY 14
D2028 CHANNEL  ; MEMORY 15
D2030 CHANNEL  ; MEMORY 16
D2032 CHANNEL  ; MEMORY 17
D2034 CHANNEL  ; MEMORY 18
D2036 CHANNEL  ; MEMORY 19
D2038 CHANNEL  ; MEMORY 20
D2040 CHANNEL  ; MEMORY 21
D2042 CHANNEL  ; MEMORY 22
D2044 CHANNEL  ; MEMORY 23
D2046 CHANNEL  ; MEMORY 24
D2048 CHANNEL  ; MEMORY 25
D2050 CHANNEL  ; MEMORY 26
D2052 CHANNEL  ; MEMORY 27
D2054 CHANNEL  ; MEMORY 28
D2056 CHANNEL  ; MEMORY 29
D2058 CHANNEL  ; MEMORY 30
D2060 CHANNEL  ; MEMORY 31
D2062 CHANNEL  ; MEMORY 32
D2064 CHANNEL  ; MEMORY 33
D2066 CHANNEL  ; MEMORY 34
D2068 CHANNEL  ; MEMORY 35
D2070 CHANNEL  ; MEMORY 36
D2072 CHANNEL  ; MEMORY 37
D2074 CHANNEL  ; MEMORY 38
D2076 CHANNEL  ; MEMORY 39
D2078 CHANNEL  ; MEMORY 40
D2080 CHANNEL  ; MEMORY 41
D2082 CHANNEL  ; MEMORY 42
D2084 CHANNEL  ; MEMORY 43
D2086 CHANNEL  ; MEMORY 44
D2088 CHANNEL  ; MEMORY 45
D2090 CHANNEL  ; MEMORY 46
D2092 CHANNEL  ; MEMORY 47
D2094 CHANNEL  ; MEMORY 48
D2096 CHANNEL  ; MEMORY 49
D2098 CHANNEL  ; MEMORY 50
D240 CHANNEL  ; DISPLAY TEACH RFID 2
D30 CHANNEL  ; TEACH RFID 4
D300 CHANNEL  ; INPUT DATA READER 2
D3000 CHANNEL  ; MEMORY 1
D3002 CHANNEL  ; MEMORY 2
D3004 CHANNEL  ; MEMORY 3
D3006 CHANNEL  ; MEMORY 4
D3008 CHANNEL  ; MEMORY 5
D3010 CHANNEL  ; MEMORY 6
D3012 CHANNEL  ; MEMORY 7
D3014 CHANNEL  ; MEMORY 8
D3016 CHANNEL  ; MEMORY 9
D3018 CHANNEL  ; MEMORY 10
D3020 CHANNEL  ; MEMORY 11
D3022 CHANNEL  ; MEMORY 12
D3024 CHANNEL  ; MEMORY 13
D3026 CHANNEL  ; MEMORY 14
D3028 CHANNEL  ; MEMORY 15
D3030 CHANNEL  ; MEMORY 16
D3032 CHANNEL  ; MEMORY 17
D3034 CHANNEL  ; MEMORY 18
D3036 CHANNEL  ; MEMORY 19
D3038 CHANNEL  ; MEMORY 20
D3040 CHANNEL  ; MEMORY 21
D3042 CHANNEL  ; MEMORY 22
D3044 CHANNEL  ; MEMORY 23
D3046 CHANNEL  ; MEMORY 24
D3048 CHANNEL  ; MEMORY 25
D3050 CHANNEL  ; MEMORY 26
D3052 CHANNEL  ; MEMORY 27
D3054 CHANNEL  ; MEMORY 28
D3056 CHANNEL  ; MEMORY 29
D3058 CHANNEL  ; MEMORY 30
D3060 CHANNEL  ; MEMORY 31
D3062 CHANNEL  ; MEMORY 32
D3064 CHANNEL  ; MEMORY 33
D3066 CHANNEL  ; MEMORY 34
D3068 CHANNEL  ; MEMORY 35
D3070 CHANNEL  ; MEMORY 36
D3072 CHANNEL  ; MEMORY 37
D3074 CHANNEL  ; MEMORY 38
D3076 CHANNEL  ; MEMORY 39
D3078 CHANNEL  ; MEMORY 40
D3080 CHANNEL  ; MEMORY 41
D3082 CHANNEL  ; MEMORY 42
D3084 CHANNEL  ; MEMORY 43
D3086 CHANNEL  ; MEMORY 44
D3088 CHANNEL  ; MEMORY 45
D3090 CHANNEL  ; MEMORY 46
D3092 CHANNEL  ; MEMORY 47
D3094 CHANNEL  ; MEMORY 48
D3096 CHANNEL  ; MEMORY 49
D3098 CHANNEL  ; MEMORY 50
D340 CHANNEL  ; DISPLAY TEACH HMI 4
D40 CHANNEL  ; DISPLAY TEACH RFID 1
D4000 CHANNEL  ; MEMORY 1
D4002 CHANNEL  ; MEMORY 2
D4004 CHANNEL  ; MEMORY 3
D4006 CHANNEL  ; MEMORY 4
D4008 CHANNEL  ; MEMORY 5
D4010 CHANNEL  ; MEMORY 6
D4012 CHANNEL  ; MEMORY 7
D4014 CHANNEL  ; MEMORY 8
D4016 CHANNEL  ; MEMORY 9
D4018 CHANNEL  ; MEMORY 10
D4020 CHANNEL  ; MEMORY 11
D4022 CHANNEL  ; MEMORY 12
D4024 CHANNEL  ; MEMORY 13
D4026 CHANNEL  ; MEMORY 14
D4028 CHANNEL  ; MEMORY 15
D4030 CHANNEL  ; MEMORY 16
D4032 CHANNEL  ; MEMORY 17
D4034 CHANNEL  ; MEMORY 18
D4036 CHANNEL  ; MEMORY 19
D4038 CHANNEL  ; MEMORY 20
D4040 CHANNEL  ; MEMORY 21
D4042 CHANNEL  ; MEMORY 22
D4044 CHANNEL  ; MEMORY 23
D4046 CHANNEL  ; MEMORY 24
D4048 CHANNEL  ; MEMORY 25
D4050 CHANNEL  ; MEMORY 26
D4052 CHANNEL  ; MEMORY 27
D4054 CHANNEL  ; MEMORY 28
D4056 CHANNEL  ; MEMORY 29
D4058 CHANNEL  ; MEMORY 30
D4060 CHANNEL  ; MEMORY 31
D4062 CHANNEL  ; MEMORY 32
D4064 CHANNEL  ; MEMORY 33
D4066 CHANNEL  ; MEMORY 34
D4068 CHANNEL  ; MEMORY 35
D4070 CHANNEL  ; MEMORY 36
D4072 CHANNEL  ; MEMORY 37
D4074 CHANNEL  ; MEMORY 38
D4076 CHANNEL  ; MEMORY 39
D4078 CHANNEL  ; MEMORY 40
D4080 CHANNEL  ; MEMORY 41
D4082 CHANNEL  ; MEMORY 42
D4084 CHANNEL  ; MEMORY 43
D4086 CHANNEL  ; MEMORY 44
D4088 CHANNEL  ; MEMORY 45
D4090 CHANNEL  ; MEMORY 46
D4092 CHANNEL  ; MEMORY 47
D4094 CHANNEL  ; MEMORY 48
D4096 CHANNEL  ; MEMORY 49
D4098 CHANNEL  ; MEMORY 50
D440 CHANNEL  ; DISPLAY TEACH HMI 5
D50 CHANNEL  ; TEACH RFID 5
D500 CHANNEL  ; NUMBER RFID DETECT
D5000 CHANNEL  ; NUMBER RFID AUTO
D550 CHANNEL  ; HMI DESTINATION LIST 1 ROT1
D552 CHANNEL  ; HMI DESTINATION LIST 2 ROT1
D554 CHANNEL  ; HMI DESTINATION LIST 3 ROT1
D560 CHANNEL  ; HMI DESTINATION LIST 1 ROT2
D562 CHANNEL  ; HMI DESTINATION LIST 2 ROT2
D564 CHANNEL  ; HMI DESTINATION LIST 3 ROT2
D570 CHANNEL  ; HMI DESTINATION LIST 1 ROT3
D572 CHANNEL  ; HMI DESTINATION LIST 2 ROT3
D574 CHANNEL  ; HMI DESTINATION LIST 3 ROT3
D580 CHANNEL  ; HMI DESTINATION LIST 1 ROT4
D582 CHANNEL  ; HMI DESTINATION LIST 2 ROT4
D584 CHANNEL  ; HMI DESTINATION LIST 3 ROT4
D6001 CHANNEL  ; STACK TURN ROT 1
D6002 CHANNEL  ; STACK 2 TURN ROT 1
D6003 CHANNEL  ; STACK TURN ROT 1
D6005 CHANNEL  ; STACK POINTER ROT1
D6007 CHANNEL  ; ROT1 ANTRIAN 1
D6008 CHANNEL  ; ROT1 ANTRIAN 2
D6009 CHANNEL  ; ROT1 ANTRIAN 3
D600.00 BOOL  ; HMI ENABLE BY PASS TRANSFER
D601 CHANNEL  ; STACK POINTER BY PASS DESTINATION
D6014 CHANNEL  ; DATA ACTION TURN ROT 1
D6017 CHANNEL  ; DATA ACTION ROT 1
D610 CHANNEL  ; HMI BY PASS DESTINATION
D70 CHANNEL  ; HMI MATERIAL DESTINATION 1
D7000 CHANNEL  ; INISIAL TURN ROT 2
D7001 CHANNEL  ; STACK TURN ROT 2
D7003 CHANNEL  ; STACK POINTER ROT2
D7005 CHANNEL  ; ROT2 ANTRIAN 1
D7006 CHANNEL  ; ROT2 ANTRIAN 2
D7007 CHANNEL  ; ROT2 ANTRIAN 3
D7014 CHANNEL  ; DATA ACTION ROT 2
D72 CHANNEL  ; HMI MATERIAL DESTINATION 2
D80 CHANNEL  ; OUT HMI DISPLAY NO RFID
D8001 CHANNEL  ; STACK TURN ROT 3
D8003 CHANNEL  ; STACK POINTER ROT3
D8005 CHANNEL  ; ROT3 ANTRIAN 1
D8006 CHANNEL  ; ROT3 ANTRIAN 2
D8007 CHANNEL  ; ROT3 ANTRIAN 3
D8014 CHANNEL  ; DATA ACTION TURN ROT 3
D9000 CHANNEL  ; RFID NUMBER ERROR1
D9001 CHANNEL  ; STACK TURN ROT 4
D9003 CHANNEL  ; STACK POINTER ROT4
D9005 CHANNEL  ; ROT4 ANTRIAN 1
D9006 CHANNEL  ; ROT4 ANTRIAN 2
D9007 CHANNEL  ; ROT4 ANTRIAN 3
D9014 CHANNEL  ; DATA ACTION ROT 4
D9100 CHANNEL  ; RFID NUMBER ERROR2
D9200 CHANNEL  ; RFID NUMBER ERROR3
T0000 BOOL  ; DELAY STP10 DOWN
T0002 BOOL  ; DELAY DOWN STP11
T0003 BOOL  ; DELAY BEFORE TRANSFER OUT M10
T0004 BOOL  ; DELAY OFF OUT ROLL 1 TURN
T0005 BOOL  ; DELAY DOWN STP13 IN
T0006 BOOL  ; DELAY M10 FWD OUT MATERIAL
T0008 BOOL  ; DELAY OUT MATERIAL
T0009 BOOL  ; DELAY OUT MATERIAL M3
T0010 BOOL  ; DELAY MOVE 99
T0011 BOOL  ; DELAY INCREMENT PHS 1
T0012 BOOL  ; DELAY DECREMENT PHS 2
T0013 BOOL  ; TIMER ALARM RFID NOT DETECT
T0014 BOOL  ; BYPASS TIMER ALARM RFID NOT DETECT
T0023 BOOL  ; DELAY MROLLER 5 OFF
T0024 BOOL  ; DELAY PH23 AFTER OFF
T0025 BOOL  ; DELAY PH2 AFTER OFF
T0026 BOOL  ; DELAY PH4 AFTER OFF
T0027 BOOL  ; DELAY PH8 AFTER OFF
T0028 BOOL  ; DELAY PH12 AFTER OFF
T0029 BOOL  ; DELAY PH16 AFTER OFF
T0030 BOOL  ; DELAY PH6 AFTER OFF
T0031 BOOL  ; DELAY PH10 AFTER OFF
T0032 BOOL  ; DELAY PH6 AFTER OFF
T0033 BOOL  ; DELAY PH18 AFTER OFF
T0034 BOOL  ; TIMEOUT M10 IN
T0035 BOOL  ; TIMEOUT MROL5 IN
T0036 BOOL  ; TIMEOUT M9 IN
T0037 BOOL  ; TIMEOUT M7 IN
T0038 BOOL  ; TIMEOUT M5 IN
T0039 BOOL  ; TIMEOUT M3 IN
T0040 BOOL  ; TIMEOUT M1 IN
T0041 BOOL  ; TIMER STOPPER DOWN ALL
T0042 BOOL  ; TIMER STP 14 DOWN
T0043 BOOL  ; DELAY PINLOCK ROT 4 UP
T0044 BOOL  ; DELAY PINLOCK ROT 3 UP
T0045 BOOL  ; DELAY PINLOCK ROT 2 UP
T0046 BOOL  ; DELAY PINLOCK ROT 1 UP
W10 CHANNEL  ; NEXT/PREV MANUAL SCREEN
W11 CHANNEL  ; NEXT MAN2
W12 CHANNEL  ; NEXT MAN3
W13 CHANNEL  ; NEXT MAN4
W14 CHANNEL  ; NEXT MAN5
W15 CHANNEL  ; NEXT MAN6
W16 CHANNEL  ; NUMBER OF SCREEN HMI
W17 CHANNEL  ; MANUAL
W18 CHANNEL  ; FAULT
W19 CHANNEL  ; SETTING
W1.04 BOOL  ; HMI OUT INDI RUN M10
W1.05 BOOL  ; HMI OUT INDI RUN M9
W1.06 BOOL  ; HMI OUT INDI RUN M8
W1.07 BOOL  ; HMI OUT INDI RUN M7
W1.08 BOOL  ; HMI OUT INDI RUN M6
W1.09 BOOL  ; HMI OUT INDI RUN M5
W1.10 BOOL  ; HMI OUT INDI RUN M4
W1.11 BOOL  ; HMI OUT INDI RUN M3
RFID 3202 UINT
ROTARY_1 ROTARY
ROTARY_11 ROTARY
ROTARY_2 ROTARY
ROTARY_22 ROTARY
ROTARY_3 ROTARY
ROTARY_4 ROTARY
ROTARY_44 ROTARY
ROTARY_TABLE_1 MANUAL_ROTARY
ROTARY_TABLE_2 MANUAL_ROTARY
ROTARY_TABLE_3 MANUAL_ROTARY
ROTARY_TABLE_33 MANUAL_ROTARY
ROTARY_TABLE_4 MANUAL_ROTARY
ROTARY_TABLE_44 MANUAL_ROTARY
SEQ_RFID_1 RFID_SEQUENCE
SEQ_RFID_2 RFID_SEQUENCE
SEQ_RFID_3 RFID_SEQUENCE
SEQ_RFID_4 RFID_SEQUENCE
SEQ_RFID_5 RFID_SEQUENCE

## Program AFTER_PAINTING (cyclic task 0)
Local symbols
F500 CHANNEL
HEX UINT
P_ON BOOL

### Section MANUAL_MODE

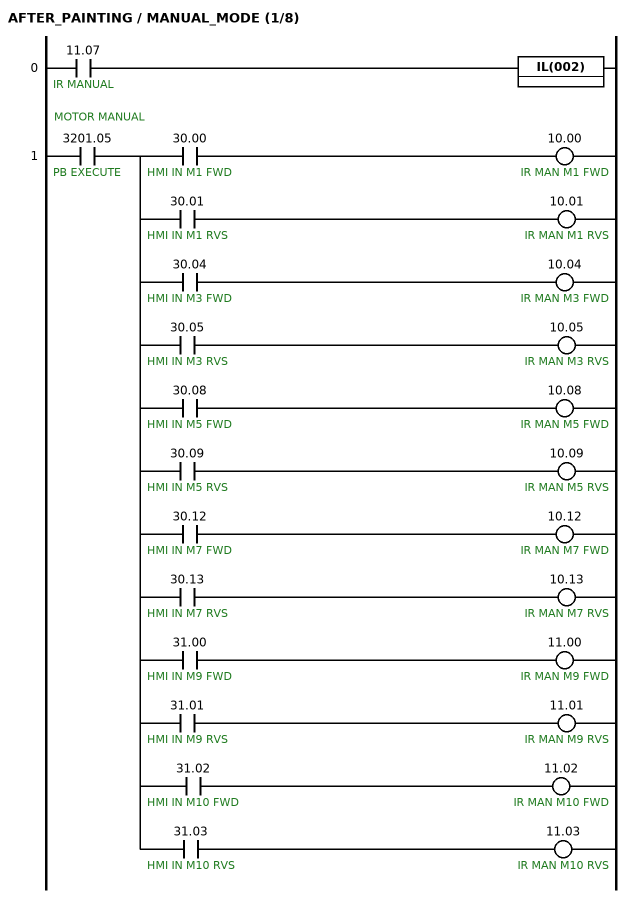
; rung 0
LD 11.07  ; IR MANUAL
IL(002)
; rung 1: MOTOR MANUAL
LD 3201.05  ; PB EXECUTE
OUT TR0
AND 30.00  ; HMI IN M1 FWD
OUT 10.00  ; IR MAN M1 FWD
LD TR0
AND 30.01  ; HMI IN M1 RVS
OUT 10.01  ; IR MAN M1 RVS
LD TR0
AND 30.04  ; HMI IN M3 FWD
OUT 10.04  ; IR MAN M3 FWD
LD TR0
AND 30.05  ; HMI IN M3 RVS
OUT 10.05  ; IR MAN M3 RVS
LD TR0
AND 30.08  ; HMI IN M5 FWD
OUT 10.08  ; IR MAN M5 FWD
LD TR0
AND 30.09  ; HMI IN M5 RVS
OUT 10.09  ; IR MAN M5 RVS
LD TR0
AND 30.12  ; HMI IN M7 FWD
OUT 10.12  ; IR MAN M7 FWD
LD TR0
AND 30.13  ; HMI IN M7 RVS
OUT 10.13  ; IR MAN M7 RVS
LD TR0
AND 31.00  ; HMI IN M9 FWD
OUT 11.00  ; IR MAN M9 FWD
LD TR0
AND 31.01  ; HMI IN M9 RVS
OUT 11.01  ; IR MAN M9 RVS
LD TR0
AND 31.02  ; HMI IN M10 FWD
OUT 11.02  ; IR MAN M10 FWD
LD TR0
AND 31.03  ; HMI IN M10 RVS
OUT 11.03  ; IR MAN M10 RVS

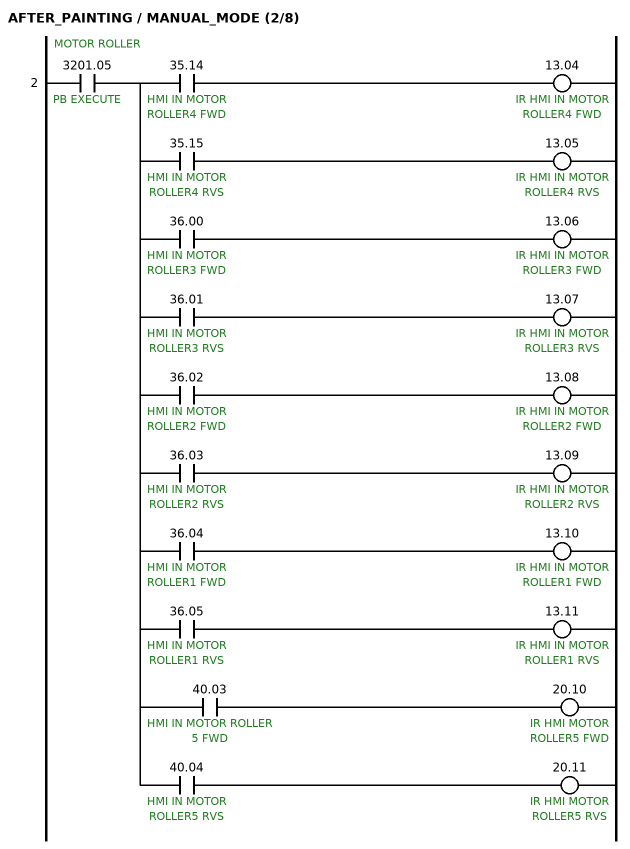
; rung 2: MOTOR ROLLER
LD 3201.05  ; PB EXECUTE
OUT TR0
AND 35.14  ; HMI IN MOTOR ROLLER4 FWD
OUT 13.04  ; IR HMI IN MOTOR ROLLER4 FWD
LD TR0
AND 35.15  ; HMI IN MOTOR ROLLER4 RVS
OUT 13.05  ; IR HMI IN MOTOR ROLLER4 RVS
LD TR0
AND 36.00  ; HMI IN MOTOR ROLLER3 FWD
OUT 13.06  ; IR HMI IN MOTOR ROLLER3 FWD
LD TR0
AND 36.01  ; HMI IN MOTOR ROLLER3 RVS
OUT 13.07  ; IR HMI IN MOTOR ROLLER3 RVS
LD TR0
AND 36.02  ; HMI IN MOTOR ROLLER2 FWD
OUT 13.08  ; IR HMI IN MOTOR ROLLER2 FWD
LD TR0
AND 36.03  ; HMI IN MOTOR ROLLER2 RVS
OUT 13.09  ; IR HMI IN MOTOR ROLLER2 RVS
LD TR0
AND 36.04  ; HMI IN MOTOR ROLLER1 FWD
OUT 13.10  ; IR HMI IN MOTOR ROLLER1 FWD
LD TR0
AND 36.05  ; HMI IN MOTOR ROLLER1 RVS
OUT 13.11  ; IR HMI IN MOTOR ROLLER1 RVS
LD TR0
AND 40.03  ; HMI IN MOTOR ROLLER 5 FWD
OUT 20.10  ; IR HMI MOTOR ROLLER5 FWD
LD TR0
AND 40.04  ; HMI IN MOTOR ROLLER5 RVS
OUT 20.11  ; IR HMI MOTOR ROLLER5 RVS

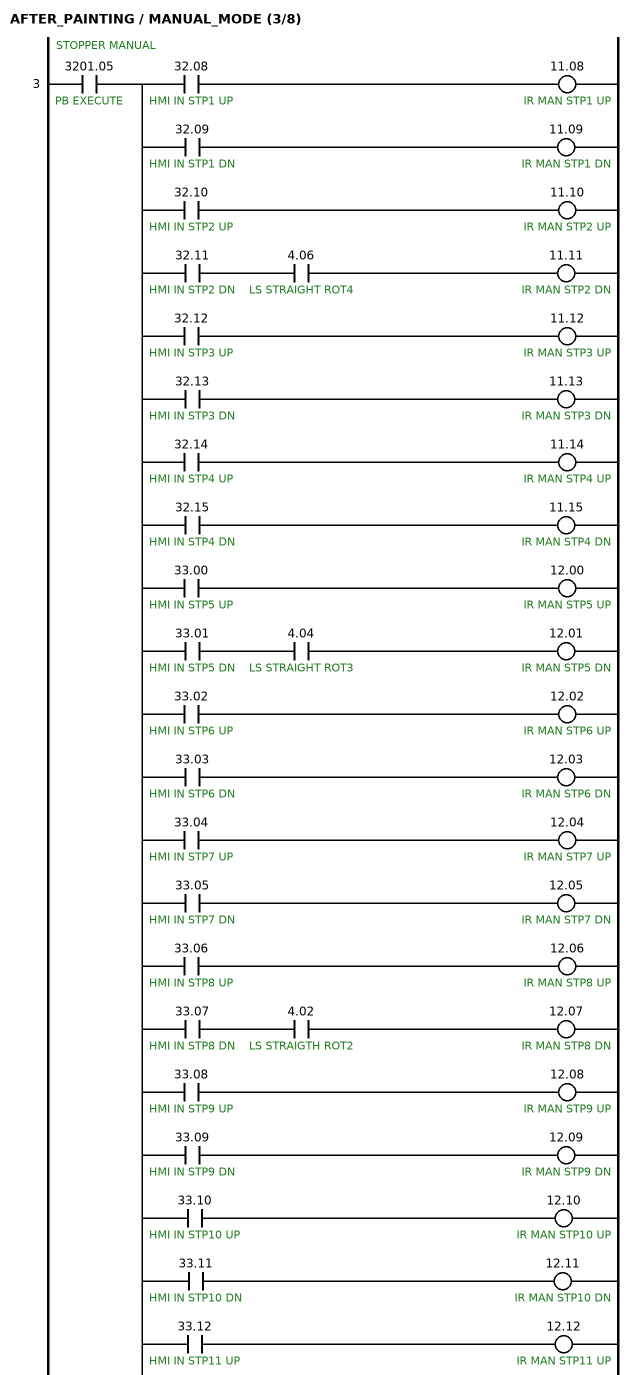

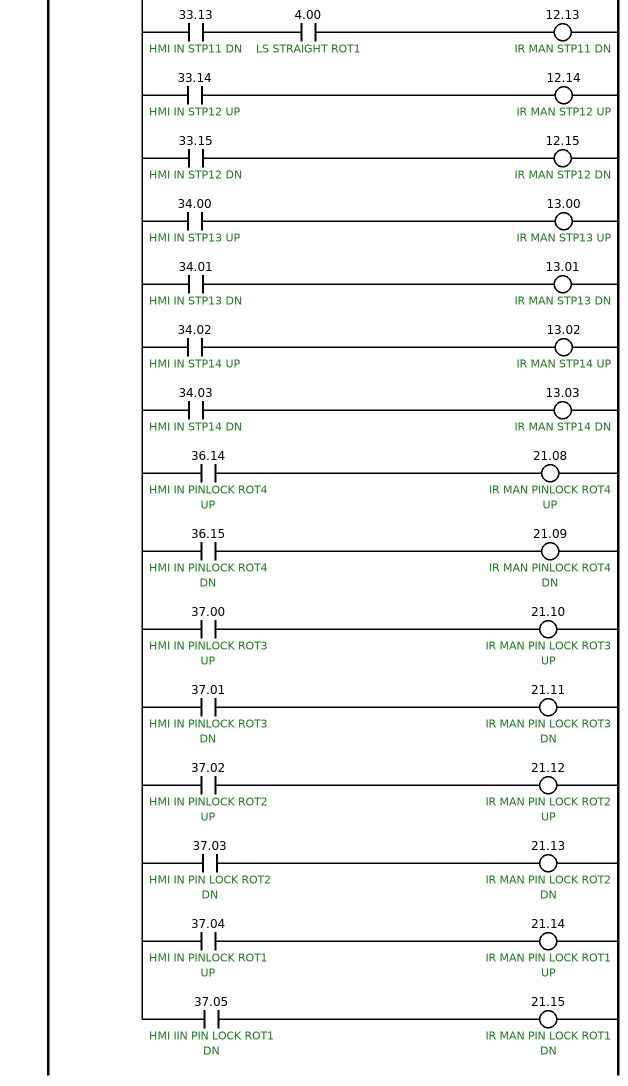
; rung 3: STOPPER MANUAL
LD 3201.05  ; PB EXECUTE
OUT TR0
AND 32.08  ; HMI IN STP1 UP
OUT 11.08  ; IR MAN STP1 UP
LD TR0
AND 32.09  ; HMI IN STP1 DN
OUT 11.09  ; IR MAN STP1 DN
LD TR0
AND 32.10  ; HMI IN STP2 UP
OUT 11.10  ; IR MAN STP2 UP
LD TR0
AND 32.11  ; HMI IN STP2 DN
AND 4.06  ; LS STRAIGHT ROT4
OUT 11.11  ; IR MAN STP2 DN
LD TR0
AND 32.12  ; HMI IN STP3 UP
OUT 11.12  ; IR MAN STP3 UP
LD TR0
AND 32.13  ; HMI IN STP3 DN
OUT 11.13  ; IR MAN STP3 DN
LD TR0
AND 32.14  ; HMI IN STP4 UP
OUT 11.14  ; IR MAN STP4 UP
LD TR0
AND 32.15  ; HMI IN STP4 DN
OUT 11.15  ; IR MAN STP4 DN
LD TR0
AND 33.00  ; HMI IN STP5 UP
OUT 12.00  ; IR MAN STP5 UP
LD TR0
AND 33.01  ; HMI IN STP5 DN
AND 4.04  ; LS STRAIGHT ROT3
OUT 12.01  ; IR MAN STP5 DN
LD TR0
AND 33.02  ; HMI IN STP6 UP
OUT 12.02  ; IR MAN STP6 UP
LD TR0
AND 33.03  ; HMI IN STP6 DN
OUT 12.03  ; IR MAN STP6 DN
LD TR0
AND 33.04  ; HMI IN STP7 UP
OUT 12.04  ; IR MAN STP7 UP
LD TR0
AND 33.05  ; HMI IN STP7 DN
OUT 12.05  ; IR MAN STP7 DN
LD TR0
AND 33.06  ; HMI IN STP8 UP
OUT 12.06  ; IR MAN STP8 UP
LD TR0
AND 33.07  ; HMI IN STP8 DN
AND 4.02  ; LS STRAIGTH ROT2
OUT 12.07  ; IR MAN STP8 DN
LD TR0
AND 33.08  ; HMI IN STP9 UP
OUT 12.08  ; IR MAN STP9 UP
LD TR0
AND 33.09  ; HMI IN STP9 DN
OUT 12.09  ; IR MAN STP9 DN
LD TR0
AND 33.10  ; HMI IN STP10 UP
OUT 12.10  ; IR MAN STP10 UP
LD TR0
AND 33.11  ; HMI IN STP10 DN
OUT 12.11  ; IR MAN STP10 DN
LD TR0
AND 33.12  ; HMI IN STP11 UP
OUT 12.12  ; IR MAN STP11 UP
LD TR0
AND 33.13  ; HMI IN STP11 DN
AND 4.00  ; LS STRAIGHT ROT1
OUT 12.13  ; IR MAN STP11 DN
LD TR0
AND 33.14  ; HMI IN STP12 UP
OUT 12.14  ; IR MAN STP12 UP
LD TR0
AND 33.15  ; HMI IN STP12 DN
OUT 12.15  ; IR MAN STP12 DN
LD TR0
AND 34.00  ; HMI IN STP13 UP
OUT 13.00  ; IR MAN STP13 UP
LD TR0
AND 34.01  ; HMI IN STP13 DN
OUT 13.01  ; IR MAN STP13 DN
LD TR0
AND 34.02  ; HMI IN STP14 UP
OUT 13.02  ; IR MAN STP14 UP
LD TR0
AND 34.03  ; HMI IN STP14 DN
OUT 13.03  ; IR MAN STP14 DN
LD TR0
AND 36.14  ; HMI IN PINLOCK ROT4 UP
OUT 21.08  ; IR MAN PINLOCK ROT4 UP
LD TR0
AND 36.15  ; HMI IN PINLOCK ROT4 DN
OUT 21.09  ; IR MAN PINLOCK ROT4 DN
LD TR0
AND 37.00  ; HMI IN PINLOCK ROT3 UP
OUT 21.10  ; IR MAN PIN LOCK ROT3 UP
LD TR0
AND 37.01  ; HMI IN PINLOCK ROT3 DN
OUT 21.11  ; IR MAN PIN LOCK ROT3 DN
LD TR0
AND 37.02  ; HMI IN PINLOCK ROT2 UP
OUT 21.12  ; IR MAN PIN LOCK ROT2 UP
LD TR0
AND 37.03  ; HMI IN PIN LOCK ROT2 DN
OUT 21.13  ; IR MAN PIN LOCK ROT2 DN
LD TR0
AND 37.04  ; HMI IN PINLOCK ROT1 UP
OUT 21.14  ; IR MAN PIN LOCK ROT1 UP
LD TR0
AND 37.05  ; HMI IIN PIN LOCK ROT1 DN
OUT 21.15  ; IR MAN PIN LOCK ROT1 DN

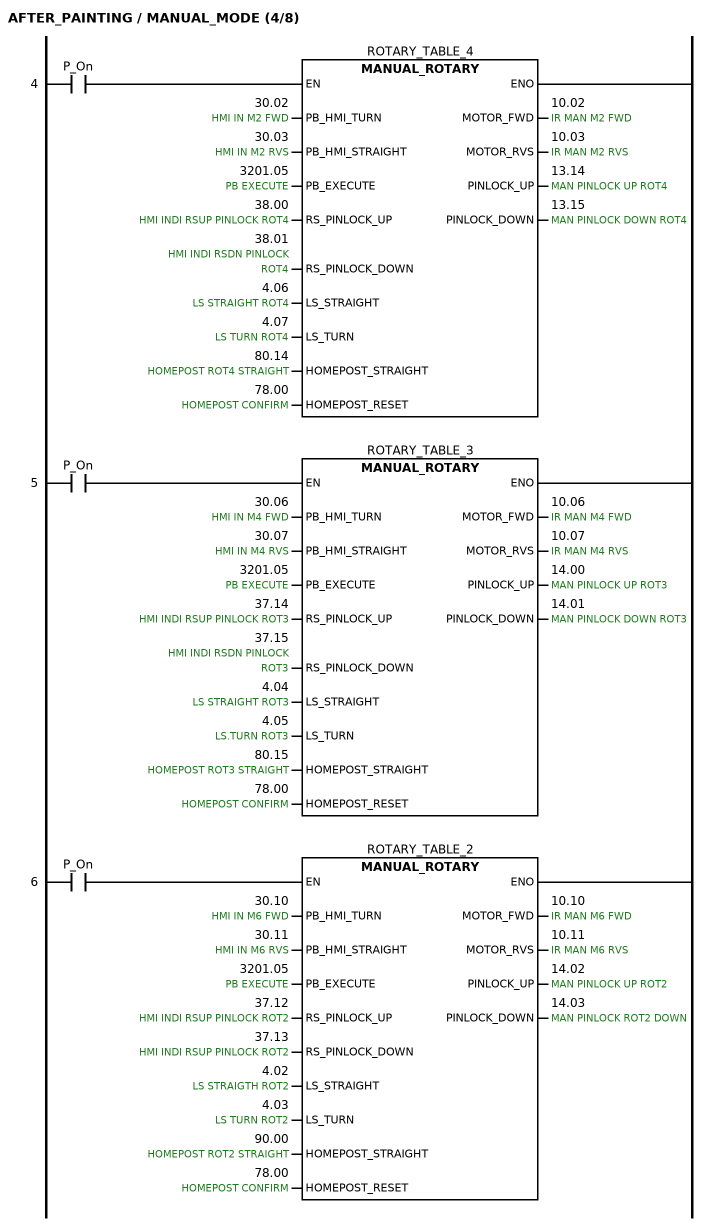
; rung 4
LD P_On
CALL ROTARY_TABLE_4 : MANUAL_ROTARY (PB_HMI_TURN := 30.02, PB_HMI_STRAIGHT := 30.03, PB_EXECUTE := 3201.05, RS_PINLOCK_UP := 38.00, RS_PINLOCK_DOWN := 38.01, LS_STRAIGHT := 4.06, LS_TURN := 4.07, HOMEPOST_STRAIGHT := 80.14, HOMEPOST_RESET := 78.00, MOTOR_FWD => 10.02, MOTOR_RVS => 10.03, PINLOCK_UP => 13.14, PINLOCK_DOWN => 13.15)  ; HMI IN M2 FWD, HMI IN M2 RVS, PB EXECUTE, HMI INDI RSUP PINLOCK ROT4, HMI INDI RSDN PINLOCK ROT4, LS STRAIGHT ROT4, LS TURN ROT4, HOMEPOST ROT4 STRAIGHT, HOMEPOST CONFIRM, IR MAN M2 FWD, IR MAN M2 RVS, MAN PINLOCK UP ROT4, MAN PINLOCK DOWN ROT4
; rung 5
LD P_On
CALL ROTARY_TABLE_3 : MANUAL_ROTARY (PB_HMI_TURN := 30.06, PB_HMI_STRAIGHT := 30.07, PB_EXECUTE := 3201.05, RS_PINLOCK_UP := 37.14, RS_PINLOCK_DOWN := 37.15, LS_STRAIGHT := 4.04, LS_TURN := 4.05, HOMEPOST_STRAIGHT := 80.15, HOMEPOST_RESET := 78.00, MOTOR_FWD => 10.06, MOTOR_RVS => 10.07, PINLOCK_UP => 14.00, PINLOCK_DOWN => 14.01)  ; HMI IN M4 FWD, HMI IN M4 RVS, PB EXECUTE, HMI INDI RSUP PINLOCK ROT3, HMI INDI RSDN PINLOCK ROT3, LS STRAIGHT ROT3, LS.TURN ROT3, HOMEPOST ROT3 STRAIGHT, HOMEPOST CONFIRM, IR MAN M4 FWD, IR MAN M4 RVS, MAN PINLOCK UP ROT3, MAN PINLOCK DOWN ROT3
; rung 6
LD P_On
CALL ROTARY_TABLE_2 : MANUAL_ROTARY (PB_HMI_TURN := 30.10, PB_HMI_STRAIGHT := 30.11, PB_EXECUTE := 3201.05, RS_PINLOCK_UP := 37.12, RS_PINLOCK_DOWN := 37.13, LS_STRAIGHT := 4.02, LS_TURN := 4.03, HOMEPOST_STRAIGHT := 90.00, HOMEPOST_RESET := 78.00, MOTOR_FWD => 10.10, MOTOR_RVS => 10.11, PINLOCK_UP => 14.02, PINLOCK_DOWN => 14.03)  ; HMI IN M6 FWD, HMI IN M6 RVS, PB EXECUTE, HMI INDI RSUP PINLOCK ROT2, LS STRAIGTH ROT2, LS TURN ROT2, HOMEPOST ROT2 STRAIGHT, HOMEPOST CONFIRM, IR MAN M6 FWD, IR MAN M6 RVS, MAN PINLOCK UP ROT2, MAN PINLOCK ROT2 DOWN

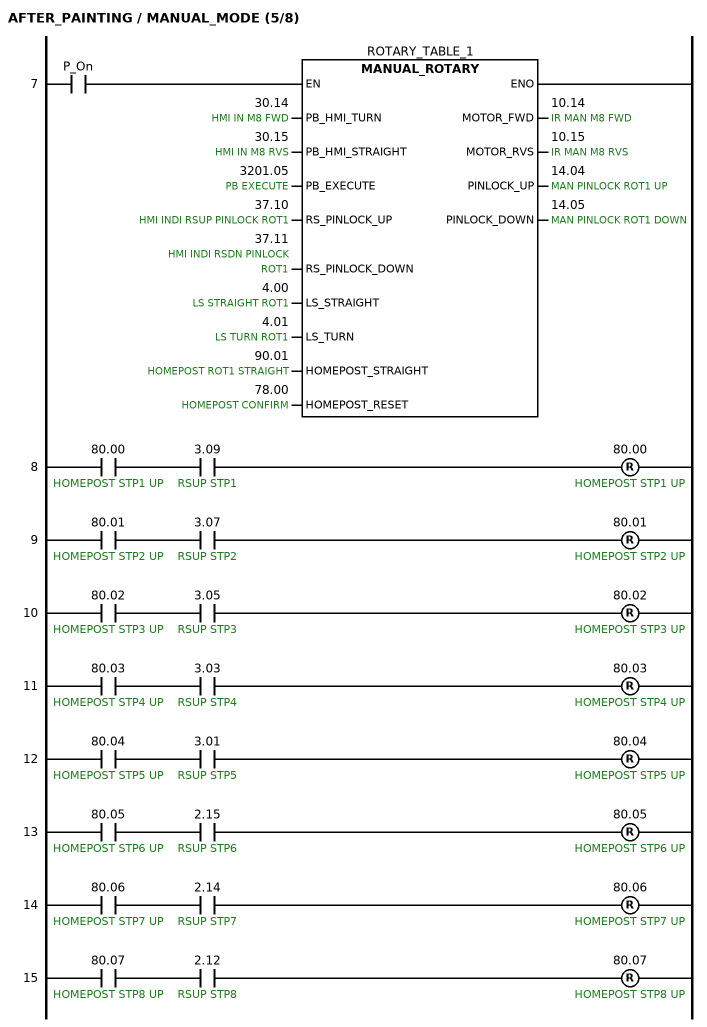
; rung 7
LD P_On
CALL ROTARY_TABLE_1 : MANUAL_ROTARY (PB_HMI_TURN := 30.14, PB_HMI_STRAIGHT := 30.15, PB_EXECUTE := 3201.05, RS_PINLOCK_UP := 37.10, RS_PINLOCK_DOWN := 37.11, LS_STRAIGHT := 4.00, LS_TURN := 4.01, HOMEPOST_STRAIGHT := 90.01, HOMEPOST_RESET := 78.00, MOTOR_FWD => 10.14, MOTOR_RVS => 10.15, PINLOCK_UP => 14.04, PINLOCK_DOWN => 14.05)  ; HMI IN M8 FWD, HMI IN M8 RVS, PB EXECUTE, HMI INDI RSUP PINLOCK ROT1, HMI INDI RSDN PINLOCK ROT1, LS STRAIGHT ROT1, LS TURN ROT1, HOMEPOST ROT1 STRAIGHT, HOMEPOST CONFIRM, IR MAN M8 FWD, IR MAN M8 RVS, MAN PINLOCK ROT1 UP, MAN PINLOCK ROT1 DOWN
; rung 8
LD 80.00  ; HOMEPOST STP1 UP
AND 3.09  ; RSUP STP1
RSET 80.00  ; HOMEPOST STP1 UP
; rung 9
LD 80.01  ; HOMEPOST STP2 UP
AND 3.07  ; RSUP STP2
RSET 80.01  ; HOMEPOST STP2 UP
; rung 10
LD 80.02  ; HOMEPOST STP3 UP
AND 3.05  ; RSUP STP3
RSET 80.02  ; HOMEPOST STP3 UP
; rung 11
LD 80.03  ; HOMEPOST STP4 UP
AND 3.03  ; RSUP STP4
RSET 80.03  ; HOMEPOST STP4 UP
; rung 12
LD 80.04  ; HOMEPOST STP5 UP
AND 3.01  ; RSUP STP5
RSET 80.04  ; HOMEPOST STP5 UP
; rung 13
LD 80.05  ; HOMEPOST STP6 UP
AND 2.15  ; RSUP STP6
RSET 80.05  ; HOMEPOST STP6 UP
; rung 14
LD 80.06  ; HOMEPOST STP7 UP
AND 2.14  ; RSUP STP7
RSET 80.06  ; HOMEPOST STP7 UP
; rung 15
LD 80.07  ; HOMEPOST STP8 UP
AND 2.12  ; RSUP STP8
RSET 80.07  ; HOMEPOST STP8 UP

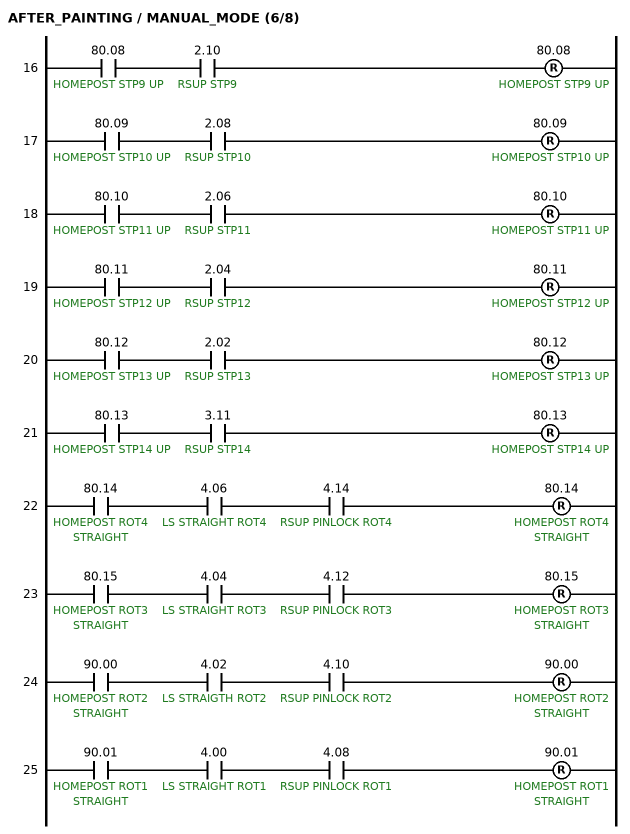
; rung 16
LD 80.08  ; HOMEPOST STP9 UP
AND 2.10  ; RSUP STP9
RSET 80.08  ; HOMEPOST STP9 UP
; rung 17
LD 80.09  ; HOMEPOST STP10 UP
AND 2.08  ; RSUP STP10
RSET 80.09  ; HOMEPOST STP10 UP
; rung 18
LD 80.10  ; HOMEPOST STP11 UP
AND 2.06  ; RSUP STP11
RSET 80.10  ; HOMEPOST STP11 UP
; rung 19
LD 80.11  ; HOMEPOST STP12 UP
AND 2.04  ; RSUP STP12
RSET 80.11  ; HOMEPOST STP12 UP
; rung 20
LD 80.12  ; HOMEPOST STP13 UP
AND 2.02  ; RSUP STP13
RSET 80.12  ; HOMEPOST STP13 UP
; rung 21
LD 80.13  ; HOMEPOST STP14 UP
AND 3.11  ; RSUP STP14
RSET 80.13  ; HOMEPOST STP14 UP
; rung 22
LD 80.14  ; HOMEPOST ROT4 STRAIGHT
AND 4.06  ; LS STRAIGHT ROT4
AND 4.14  ; RSUP PINLOCK ROT4
RSET 80.14  ; HOMEPOST ROT4 STRAIGHT
; rung 23
LD 80.15  ; HOMEPOST ROT3 STRAIGHT
AND 4.04  ; LS STRAIGHT ROT3
AND 4.12  ; RSUP PINLOCK ROT3
RSET 80.15  ; HOMEPOST ROT3 STRAIGHT
; rung 24
LD 90.00  ; HOMEPOST ROT2 STRAIGHT
AND 4.02  ; LS STRAIGTH ROT2
AND 4.10  ; RSUP PINLOCK ROT2
RSET 90.00  ; HOMEPOST ROT2 STRAIGHT
; rung 25
LD 90.01  ; HOMEPOST ROT1 STRAIGHT
AND 4.00  ; LS STRAIGHT ROT1
AND 4.08  ; RSUP PINLOCK ROT1
RSET 90.01  ; HOMEPOST ROT1 STRAIGHT

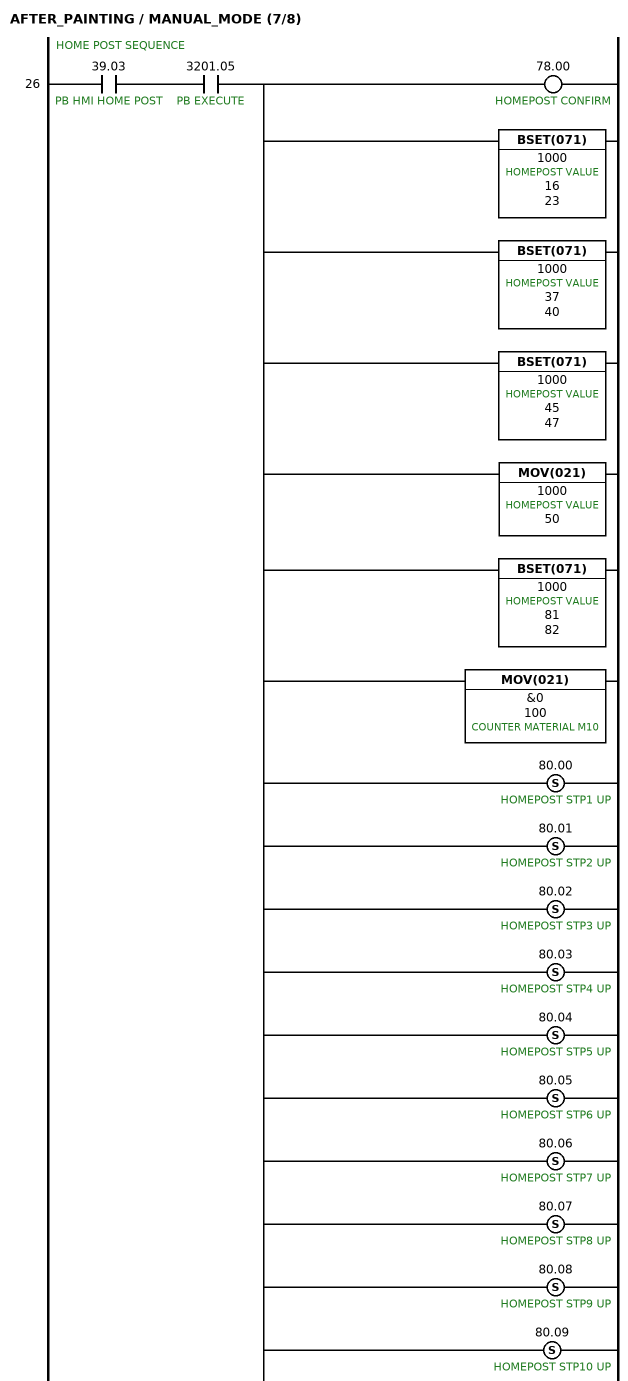

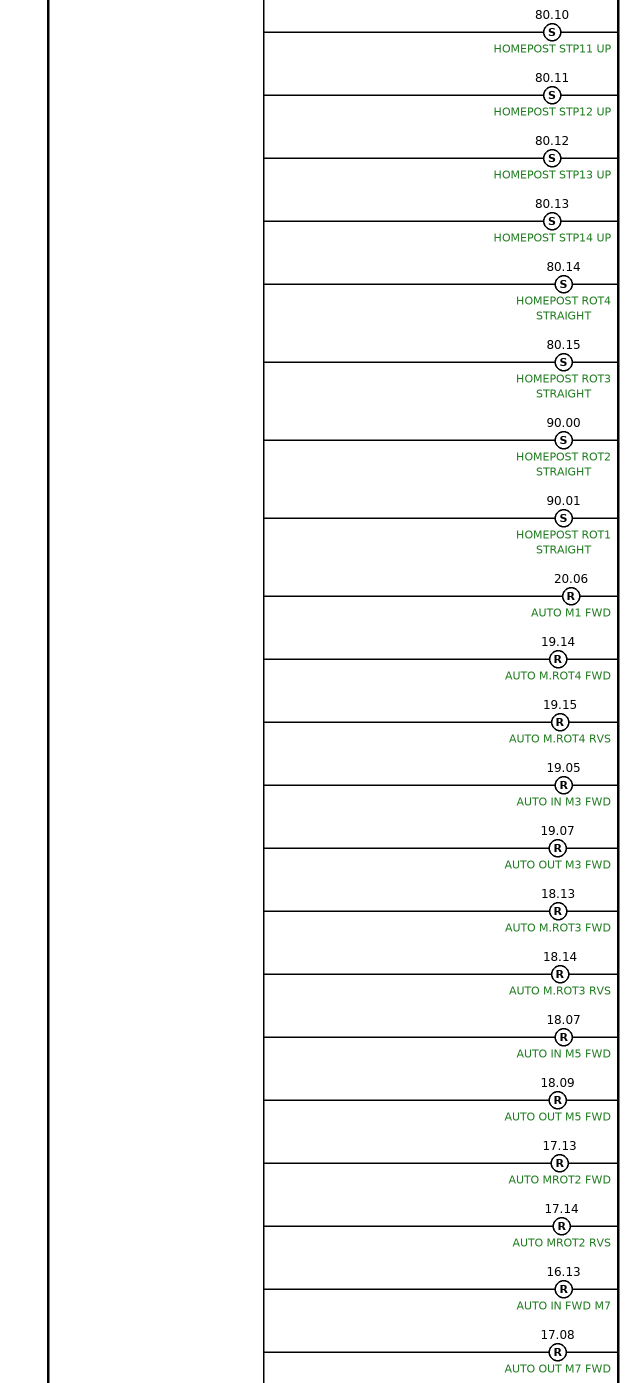

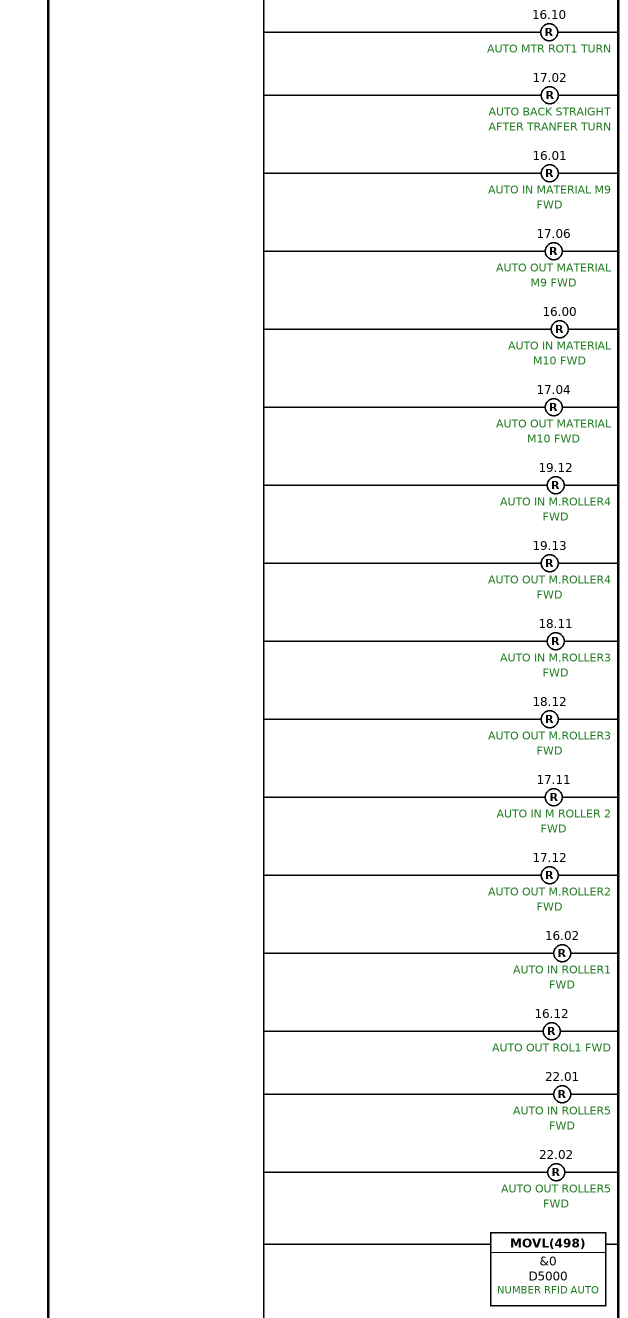

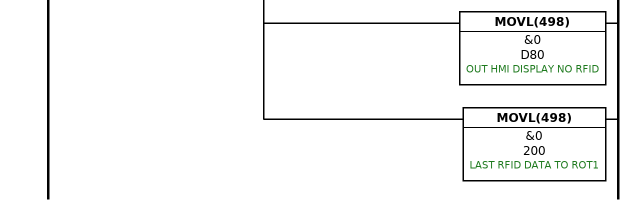
; rung 26: HOME POST SEQUENCE
LD 39.03  ; PB HMI HOME POST
AND 3201.05  ; PB EXECUTE
OUT 78.00  ; HOMEPOST CONFIRM
BSET(071) 1000 16 23  ; HOMEPOST VALUE
BSET(071) 1000 37 40  ; HOMEPOST VALUE
BSET(071) 1000 45 47  ; HOMEPOST VALUE
MOV(021) 1000 50  ; HOMEPOST VALUE
BSET(071) 1000 81 82  ; HOMEPOST VALUE
MOV(021) &0 100  ; COUNTER MATERIAL M10
SET 80.00  ; HOMEPOST STP1 UP
SET 80.01  ; HOMEPOST STP2 UP
SET 80.02  ; HOMEPOST STP3 UP
SET 80.03  ; HOMEPOST STP4 UP
SET 80.04  ; HOMEPOST STP5 UP
SET 80.05  ; HOMEPOST STP6 UP
SET 80.06  ; HOMEPOST STP7 UP
SET 80.07  ; HOMEPOST STP8 UP
SET 80.08  ; HOMEPOST STP9 UP
SET 80.09  ; HOMEPOST STP10 UP
SET 80.10  ; HOMEPOST STP11 UP
SET 80.11  ; HOMEPOST STP12 UP
SET 80.12  ; HOMEPOST STP13 UP
SET 80.13  ; HOMEPOST STP14 UP
SET 80.14  ; HOMEPOST ROT4 STRAIGHT
SET 80.15  ; HOMEPOST ROT3 STRAIGHT
SET 90.00  ; HOMEPOST ROT2 STRAIGHT
SET 90.01  ; HOMEPOST ROT1 STRAIGHT
RSET 20.06  ; AUTO M1 FWD
RSET 19.14  ; AUTO M.ROT4 FWD
RSET 19.15  ; AUTO M.ROT4 RVS
RSET 19.05  ; AUTO IN M3 FWD
RSET 19.07  ; AUTO OUT M3 FWD
RSET 18.13  ; AUTO M.ROT3 FWD
RSET 18.14  ; AUTO M.ROT3 RVS
RSET 18.07  ; AUTO IN M5 FWD
RSET 18.09  ; AUTO OUT M5 FWD
RSET 17.13  ; AUTO MROT2 FWD
RSET 17.14  ; AUTO MROT2 RVS
RSET 16.13  ; AUTO IN FWD M7
RSET 17.08  ; AUTO OUT M7 FWD
RSET 16.10  ; AUTO MTR ROT1 TURN
RSET 17.02  ; AUTO BACK STRAIGHT AFTER TRANFER TURN
RSET 16.01  ; AUTO IN MATERIAL M9 FWD
RSET 17.06  ; AUTO OUT MATERIAL M9 FWD
RSET 16.00  ; AUTO IN MATERIAL M10 FWD
RSET 17.04  ; AUTO OUT MATERIAL M10 FWD
RSET 19.12  ; AUTO IN M.ROLLER4 FWD
RSET 19.13  ; AUTO OUT M.ROLLER4 FWD
RSET 18.11  ; AUTO IN M.ROLLER3 FWD
RSET 18.12  ; AUTO OUT M.ROLLER3 FWD
RSET 17.11  ; AUTO IN M ROLLER 2 FWD
RSET 17.12  ; AUTO OUT M.ROLLER2 FWD
RSET 16.02  ; AUTO IN ROLLER1 FWD
RSET 16.12  ; AUTO OUT ROL1 FWD
RSET 22.01  ; AUTO IN ROLLER5 FWD
RSET 22.02  ; AUTO OUT ROLLER5 FWD
MOVL(498) &0 D5000  ; NUMBER RFID AUTO
MOVL(498) &0 D80  ; OUT HMI DISPLAY NO RFID
MOVL(498) &0 200  ; LAST RFID DATA TO ROT1

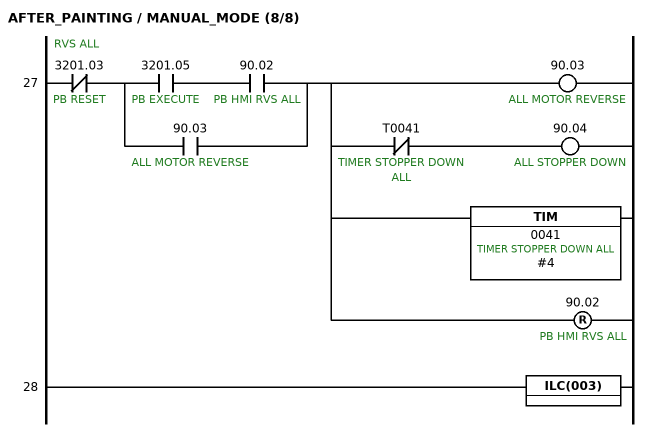
; rung 27: RVS ALL
LDNOT 3201.03  ; PB RESET
LD 3201.05  ; PB EXECUTE
AND 90.02  ; PB HMI RVS ALL
OR 90.03  ; ALL MOTOR REVERSE
ANDLD
OUT TR0
OUT 90.03  ; ALL MOTOR REVERSE
ANDNOT T0041  ; TIMER STOPPER DOWN ALL
OUT 90.04  ; ALL STOPPER DOWN
LD TR0
TIM 0041 #4  ; TIMER STOPPER DOWN ALL
RSET 90.02  ; PB HMI RVS ALL
; rung 28
ILC(003)

### Section OUTPUT_REAL

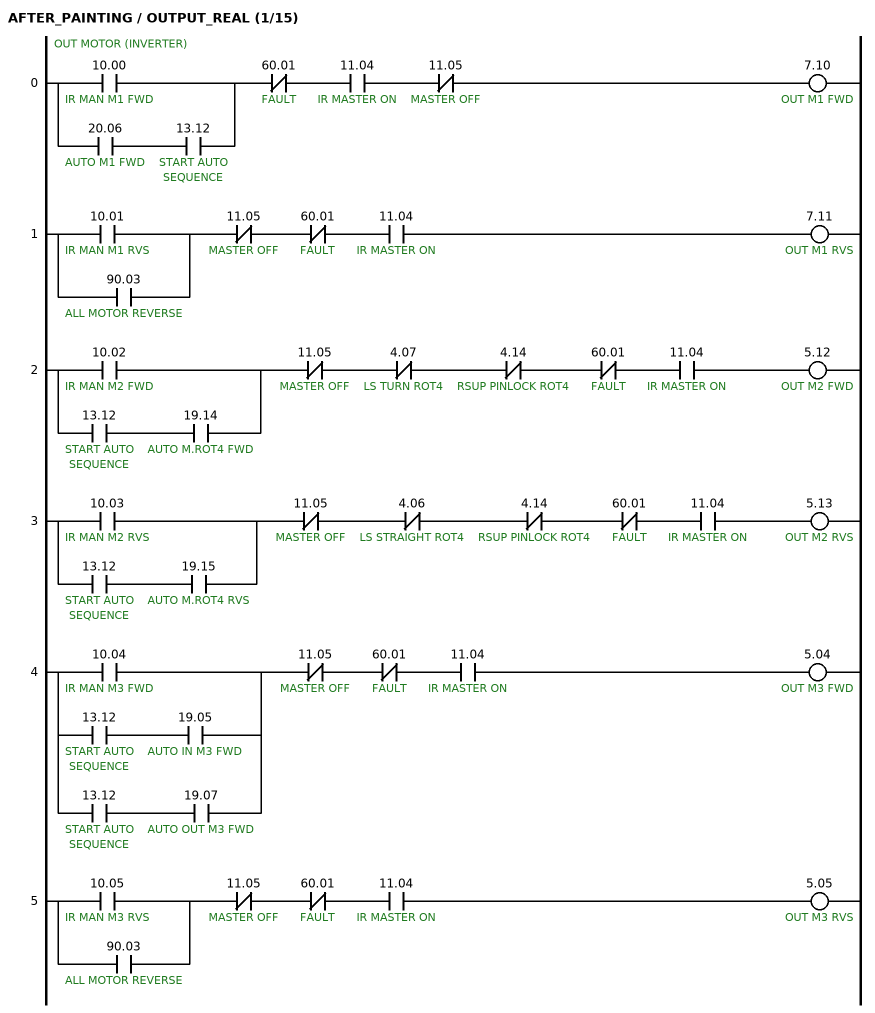
; rung 0: OUT MOTOR (INVERTER)
LD 10.00  ; IR MAN M1 FWD
LD 20.06  ; AUTO M1 FWD
AND 13.12  ; START AUTO SEQUENCE
ORLD
ANDNOT 60.01  ; FAULT
AND 11.04  ; IR MASTER ON
ANDNOT 11.05  ; MASTER OFF
OUT 7.10  ; OUT M1 FWD
; rung 1
LD 10.01  ; IR MAN M1 RVS
OR 90.03  ; ALL MOTOR REVERSE
ANDNOT 11.05  ; MASTER OFF
ANDNOT 60.01  ; FAULT
AND 11.04  ; IR MASTER ON
OUT 7.11  ; OUT M1 RVS
; rung 2
LD 10.02  ; IR MAN M2 FWD
LD 13.12  ; START AUTO SEQUENCE
AND 19.14  ; AUTO M.ROT4 FWD
ORLD
ANDNOT 11.05  ; MASTER OFF
ANDNOT 4.07  ; LS TURN ROT4
ANDNOT 4.14  ; RSUP PINLOCK ROT4
ANDNOT 60.01  ; FAULT
AND 11.04  ; IR MASTER ON
OUT 5.12  ; OUT M2 FWD
; rung 3
LD 10.03  ; IR MAN M2 RVS
LD 13.12  ; START AUTO SEQUENCE
AND 19.15  ; AUTO M.ROT4 RVS
ORLD
ANDNOT 11.05  ; MASTER OFF
ANDNOT 4.06  ; LS STRAIGHT ROT4
ANDNOT 4.14  ; RSUP PINLOCK ROT4
ANDNOT 60.01  ; FAULT
AND 11.04  ; IR MASTER ON
OUT 5.13  ; OUT M2 RVS
; rung 4
LD 10.04  ; IR MAN M3 FWD
LD 13.12  ; START AUTO SEQUENCE
AND 19.05  ; AUTO IN M3 FWD
ORLD
LD 13.12  ; START AUTO SEQUENCE
AND 19.07  ; AUTO OUT M3 FWD
ORLD
ANDNOT 11.05  ; MASTER OFF
ANDNOT 60.01  ; FAULT
AND 11.04  ; IR MASTER ON
OUT 5.04  ; OUT M3 FWD
; rung 5
LD 10.05  ; IR MAN M3 RVS
OR 90.03  ; ALL MOTOR REVERSE
ANDNOT 11.05  ; MASTER OFF
ANDNOT 60.01  ; FAULT
AND 11.04  ; IR MASTER ON
OUT 5.05  ; OUT M3 RVS

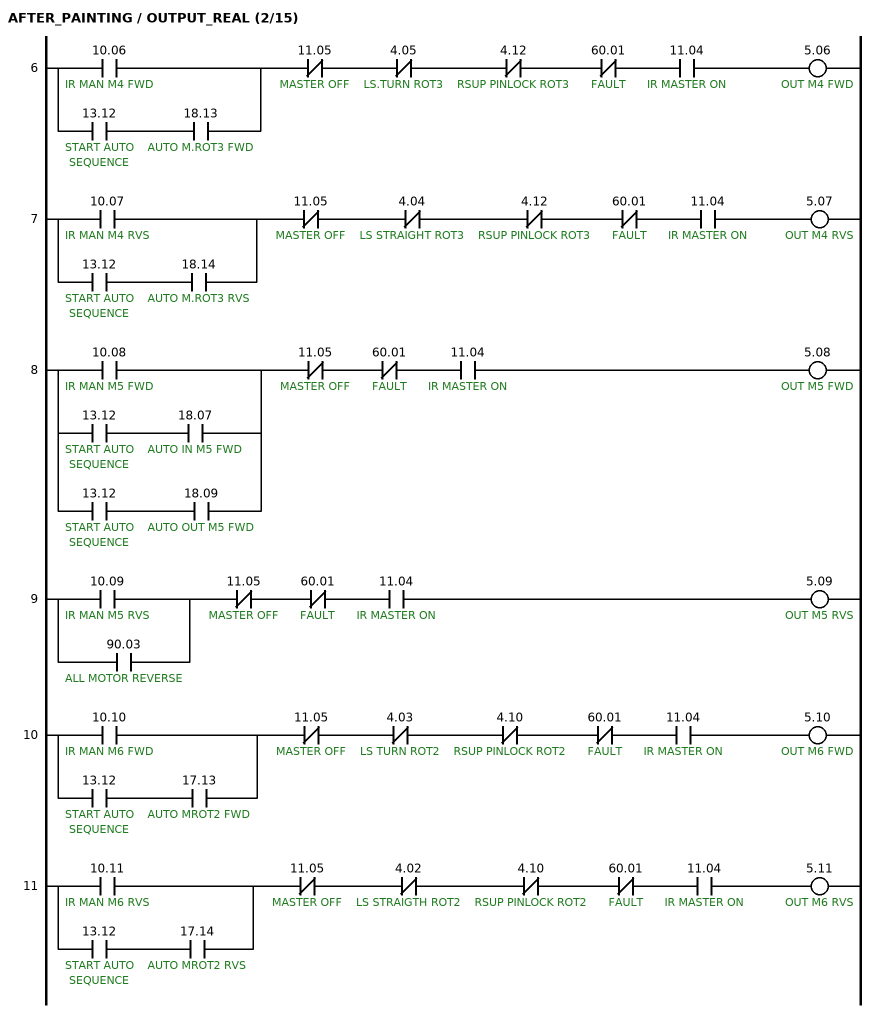
; rung 6
LD 10.06  ; IR MAN M4 FWD
LD 13.12  ; START AUTO SEQUENCE
AND 18.13  ; AUTO M.ROT3 FWD
ORLD
ANDNOT 11.05  ; MASTER OFF
ANDNOT 4.05  ; LS.TURN ROT3
ANDNOT 4.12  ; RSUP PINLOCK ROT3
ANDNOT 60.01  ; FAULT
AND 11.04  ; IR MASTER ON
OUT 5.06  ; OUT M4 FWD
; rung 7
LD 10.07  ; IR MAN M4 RVS
LD 13.12  ; START AUTO SEQUENCE
AND 18.14  ; AUTO M.ROT3 RVS
ORLD
ANDNOT 11.05  ; MASTER OFF
ANDNOT 4.04  ; LS STRAIGHT ROT3
ANDNOT 4.12  ; RSUP PINLOCK ROT3
ANDNOT 60.01  ; FAULT
AND 11.04  ; IR MASTER ON
OUT 5.07  ; OUT M4 RVS
; rung 8
LD 10.08  ; IR MAN M5 FWD
LD 13.12  ; START AUTO SEQUENCE
AND 18.07  ; AUTO IN M5 FWD
ORLD
LD 13.12  ; START AUTO SEQUENCE
AND 18.09  ; AUTO OUT M5 FWD
ORLD
ANDNOT 11.05  ; MASTER OFF
ANDNOT 60.01  ; FAULT
AND 11.04  ; IR MASTER ON
OUT 5.08  ; OUT M5 FWD
; rung 9
LD 10.09  ; IR MAN M5 RVS
OR 90.03  ; ALL MOTOR REVERSE
ANDNOT 11.05  ; MASTER OFF
ANDNOT 60.01  ; FAULT
AND 11.04  ; IR MASTER ON
OUT 5.09  ; OUT M5 RVS
; rung 10
LD 10.10  ; IR MAN M6 FWD
LD 13.12  ; START AUTO SEQUENCE
AND 17.13  ; AUTO MROT2 FWD
ORLD
ANDNOT 11.05  ; MASTER OFF
ANDNOT 4.03  ; LS TURN ROT2
ANDNOT 4.10  ; RSUP PINLOCK ROT2
ANDNOT 60.01  ; FAULT
AND 11.04  ; IR MASTER ON
OUT 5.10  ; OUT M6 FWD
; rung 11
LD 10.11  ; IR MAN M6 RVS
LD 13.12  ; START AUTO SEQUENCE
AND 17.14  ; AUTO MROT2 RVS
ORLD
ANDNOT 11.05  ; MASTER OFF
ANDNOT 4.02  ; LS STRAIGTH ROT2
ANDNOT 4.10  ; RSUP PINLOCK ROT2
ANDNOT 60.01  ; FAULT
AND 11.04  ; IR MASTER ON
OUT 5.11  ; OUT M6 RVS

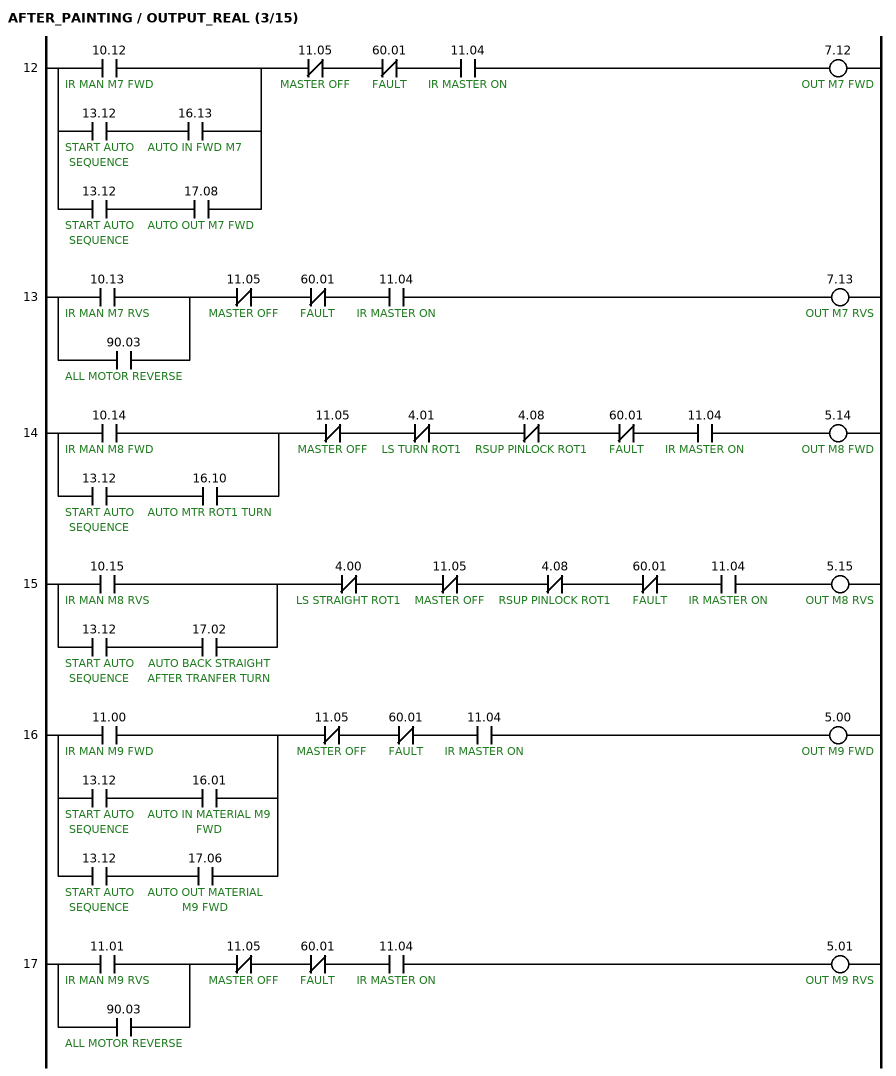
; rung 12
LD 10.12  ; IR MAN M7 FWD
LD 13.12  ; START AUTO SEQUENCE
AND 16.13  ; AUTO IN FWD M7
ORLD
LD 13.12  ; START AUTO SEQUENCE
AND 17.08  ; AUTO OUT M7 FWD
ORLD
ANDNOT 11.05  ; MASTER OFF
ANDNOT 60.01  ; FAULT
AND 11.04  ; IR MASTER ON
OUT 7.12  ; OUT M7 FWD
; rung 13
LD 10.13  ; IR MAN M7 RVS
OR 90.03  ; ALL MOTOR REVERSE
ANDNOT 11.05  ; MASTER OFF
ANDNOT 60.01  ; FAULT
AND 11.04  ; IR MASTER ON
OUT 7.13  ; OUT M7 RVS
; rung 14
LD 10.14  ; IR MAN M8 FWD
LD 13.12  ; START AUTO SEQUENCE
AND 16.10  ; AUTO MTR ROT1 TURN
ORLD
ANDNOT 11.05  ; MASTER OFF
ANDNOT 4.01  ; LS TURN ROT1
ANDNOT 4.08  ; RSUP PINLOCK ROT1
ANDNOT 60.01  ; FAULT
AND 11.04  ; IR MASTER ON
OUT 5.14  ; OUT M8 FWD
; rung 15
LD 10.15  ; IR MAN M8 RVS
LD 13.12  ; START AUTO SEQUENCE
AND 17.02  ; AUTO BACK STRAIGHT AFTER TRANFER TURN
ORLD
ANDNOT 4.00  ; LS STRAIGHT ROT1
ANDNOT 11.05  ; MASTER OFF
ANDNOT 4.08  ; RSUP PINLOCK ROT1
ANDNOT 60.01  ; FAULT
AND 11.04  ; IR MASTER ON
OUT 5.15  ; OUT M8 RVS
; rung 16
LD 11.00  ; IR MAN M9 FWD
LD 13.12  ; START AUTO SEQUENCE
AND 16.01  ; AUTO IN MATERIAL M9 FWD
ORLD
LD 13.12  ; START AUTO SEQUENCE
AND 17.06  ; AUTO OUT MATERIAL M9 FWD
ORLD
ANDNOT 11.05  ; MASTER OFF
ANDNOT 60.01  ; FAULT
AND 11.04  ; IR MASTER ON
OUT 5.00  ; OUT M9 FWD
; rung 17
LD 11.01  ; IR MAN M9 RVS
OR 90.03  ; ALL MOTOR REVERSE
ANDNOT 11.05  ; MASTER OFF
ANDNOT 60.01  ; FAULT
AND 11.04  ; IR MASTER ON
OUT 5.01  ; OUT M9 RVS

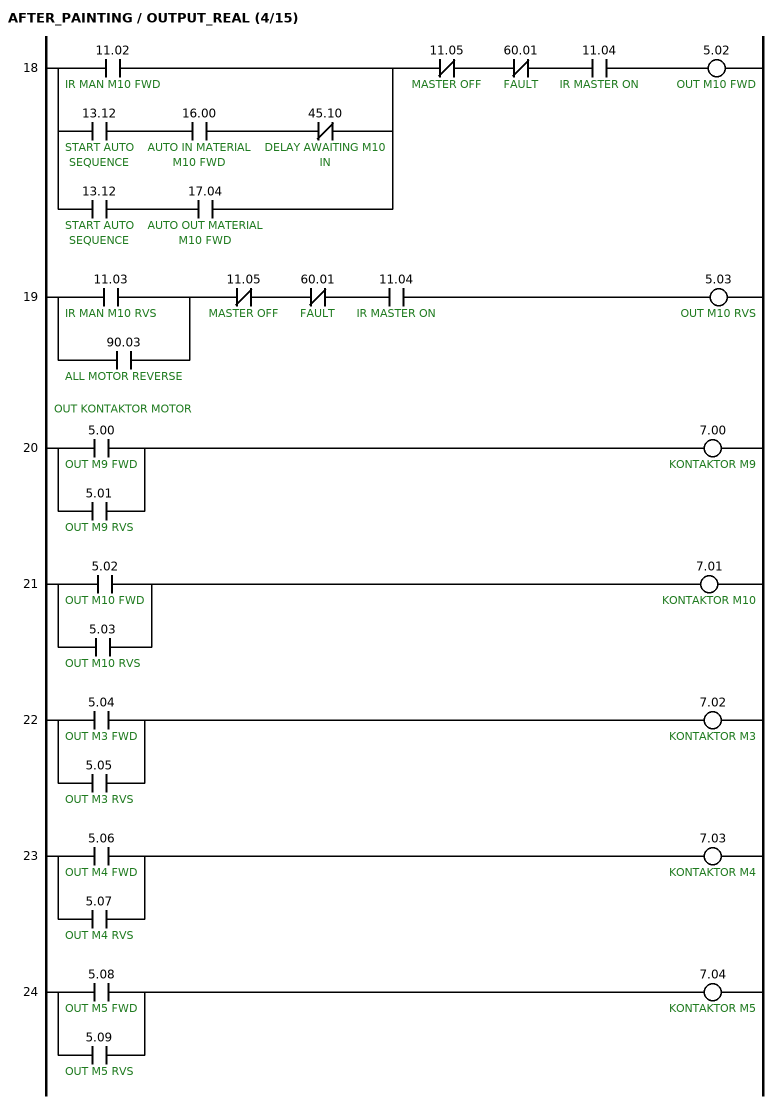
; rung 18
LD 11.02  ; IR MAN M10 FWD
LD 13.12  ; START AUTO SEQUENCE
AND 16.00  ; AUTO IN MATERIAL M10 FWD
ANDNOT 45.10  ; DELAY AWAITING M10 IN
ORLD
LD 13.12  ; START AUTO SEQUENCE
AND 17.04  ; AUTO OUT MATERIAL M10 FWD
ORLD
ANDNOT 11.05  ; MASTER OFF
ANDNOT 60.01  ; FAULT
AND 11.04  ; IR MASTER ON
OUT 5.02  ; OUT M10 FWD
; rung 19
LD 11.03  ; IR MAN M10 RVS
OR 90.03  ; ALL MOTOR REVERSE
ANDNOT 11.05  ; MASTER OFF
ANDNOT 60.01  ; FAULT
AND 11.04  ; IR MASTER ON
OUT 5.03  ; OUT M10 RVS
; rung 20: OUT KONTAKTOR MOTOR
LD 5.00  ; OUT M9 FWD
OR 5.01  ; OUT M9 RVS
OUT 7.00  ; KONTAKTOR M9
; rung 21
LD 5.02  ; OUT M10 FWD
OR 5.03  ; OUT M10 RVS
OUT 7.01  ; KONTAKTOR M10
; rung 22
LD 5.04  ; OUT M3 FWD
OR 5.05  ; OUT M3 RVS
OUT 7.02  ; KONTAKTOR M3
; rung 23
LD 5.06  ; OUT M4 FWD
OR 5.07  ; OUT M4 RVS
OUT 7.03  ; KONTAKTOR M4
; rung 24
LD 5.08  ; OUT M5 FWD
OR 5.09  ; OUT M5 RVS
OUT 7.04  ; KONTAKTOR M5

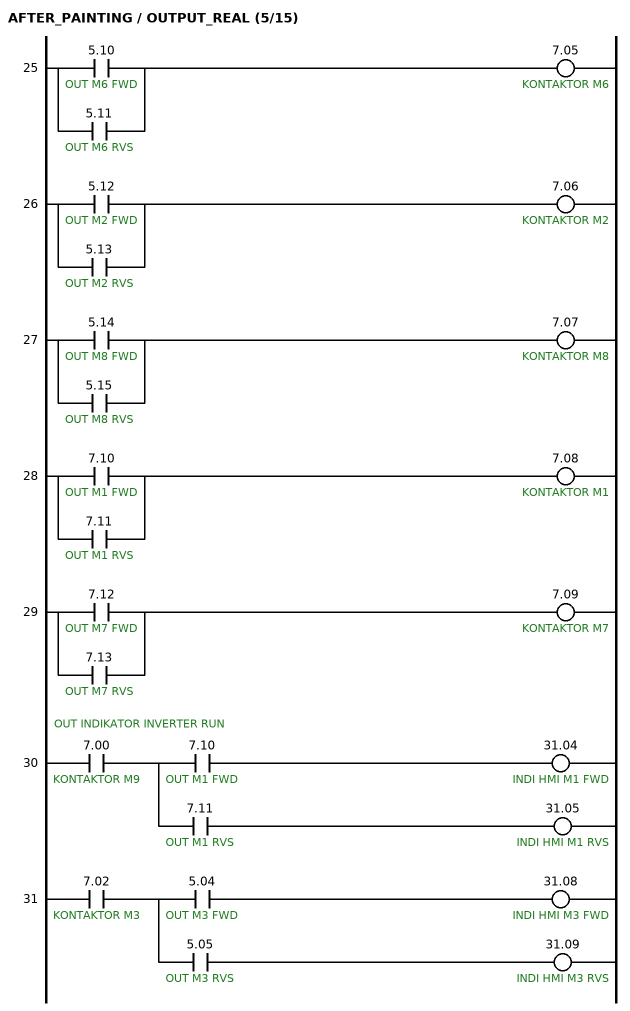
; rung 25
LD 5.10  ; OUT M6 FWD
OR 5.11  ; OUT M6 RVS
OUT 7.05  ; KONTAKTOR M6
; rung 26
LD 5.12  ; OUT M2 FWD
OR 5.13  ; OUT M2 RVS
OUT 7.06  ; KONTAKTOR M2
; rung 27
LD 5.14  ; OUT M8 FWD
OR 5.15  ; OUT M8 RVS
OUT 7.07  ; KONTAKTOR M8
; rung 28
LD 7.10  ; OUT M1 FWD
OR 7.11  ; OUT M1 RVS
OUT 7.08  ; KONTAKTOR M1
; rung 29
LD 7.12  ; OUT M7 FWD
OR 7.13  ; OUT M7 RVS
OUT 7.09  ; KONTAKTOR M7
; rung 30: OUT INDIKATOR INVERTER RUN
LD 7.00  ; KONTAKTOR M9
OUT TR0
AND 7.10  ; OUT M1 FWD
OUT 31.04  ; INDI HMI M1 FWD
LD TR0
AND 7.11  ; OUT M1 RVS
OUT 31.05  ; INDI HMI M1 RVS
; rung 31
LD 7.02  ; KONTAKTOR M3
OUT TR0
AND 5.04  ; OUT M3 FWD
OUT 31.08  ; INDI HMI M3 FWD
LD TR0
AND 5.05  ; OUT M3 RVS
OUT 31.09  ; INDI HMI M3 RVS

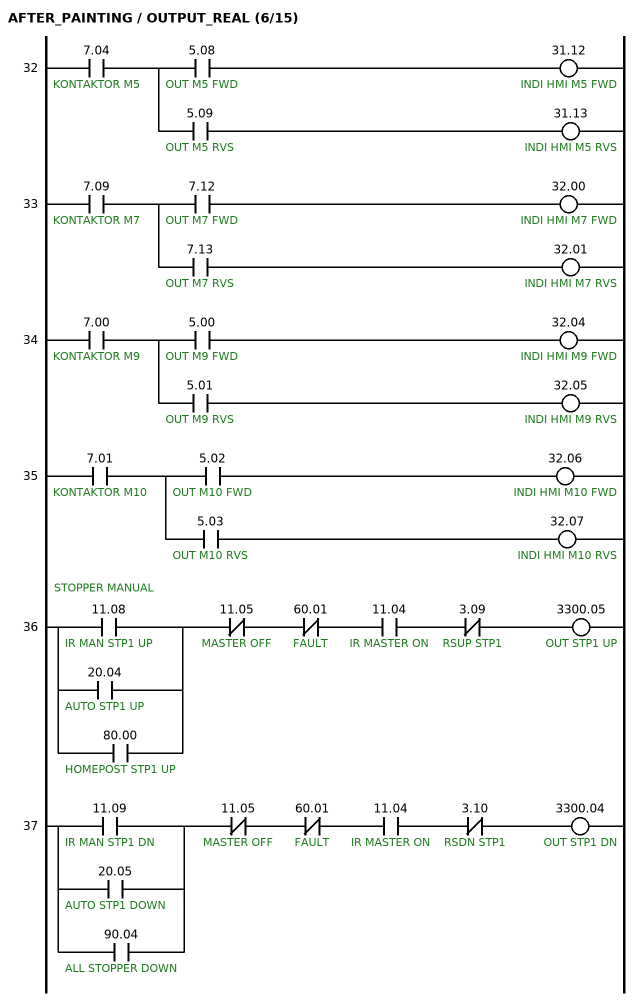
; rung 32
LD 7.04  ; KONTAKTOR M5
OUT TR0
AND 5.08  ; OUT M5 FWD
OUT 31.12  ; INDI HMI M5 FWD
LD TR0
AND 5.09  ; OUT M5 RVS
OUT 31.13  ; INDI HMI M5 RVS
; rung 33
LD 7.09  ; KONTAKTOR M7
OUT TR0
AND 7.12  ; OUT M7 FWD
OUT 32.00  ; INDI HMI M7 FWD
LD TR0
AND 7.13  ; OUT M7 RVS
OUT 32.01  ; INDI HMI M7 RVS
; rung 34
LD 7.00  ; KONTAKTOR M9
OUT TR0
AND 5.00  ; OUT M9 FWD
OUT 32.04  ; INDI HMI M9 FWD
LD TR0
AND 5.01  ; OUT M9 RVS
OUT 32.05  ; INDI HMI M9 RVS
; rung 35
LD 7.01  ; KONTAKTOR M10
OUT TR0
AND 5.02  ; OUT M10 FWD
OUT 32.06  ; INDI HMI M10 FWD
LD TR0
AND 5.03  ; OUT M10 RVS
OUT 32.07  ; INDI HMI M10 RVS
; rung 36: STOPPER MANUAL
LD 11.08  ; IR MAN STP1 UP
OR 20.04  ; AUTO STP1 UP
OR 80.00  ; HOMEPOST STP1 UP
ANDNOT 11.05  ; MASTER OFF
ANDNOT 60.01  ; FAULT
AND 11.04  ; IR MASTER ON
ANDNOT 3.09  ; RSUP STP1
OUT 3300.05  ; OUT STP1 UP
; rung 37
LD 11.09  ; IR MAN STP1 DN
OR 20.05  ; AUTO STP1 DOWN
OR 90.04  ; ALL STOPPER DOWN
ANDNOT 11.05  ; MASTER OFF
ANDNOT 60.01  ; FAULT
AND 11.04  ; IR MASTER ON
ANDNOT 3.10  ; RSDN STP1
OUT 3300.04  ; OUT STP1 DN

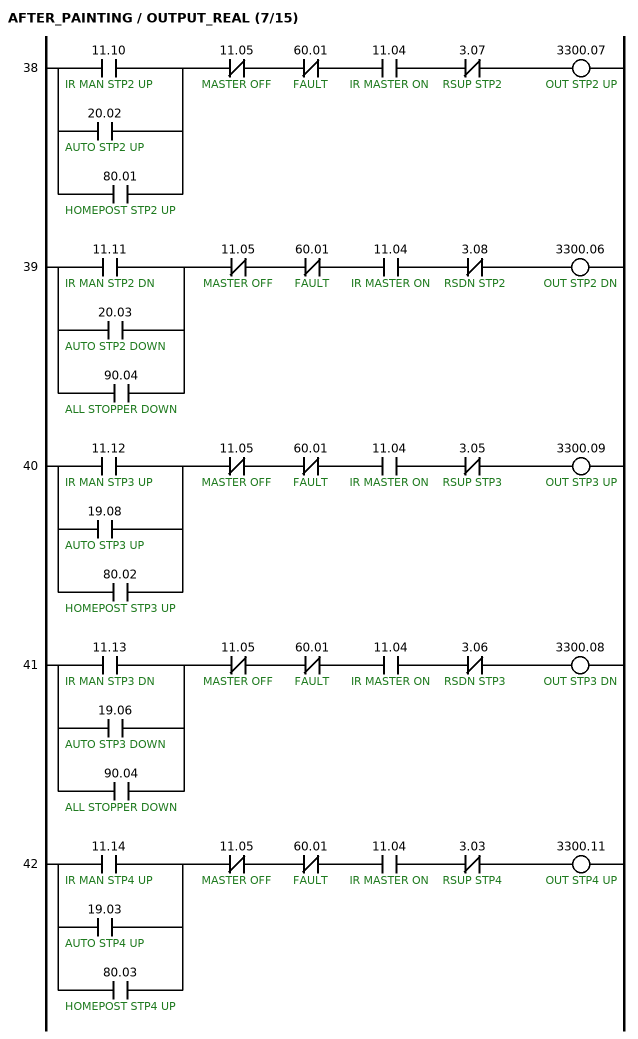
; rung 38
LD 11.10  ; IR MAN STP2 UP
OR 20.02  ; AUTO STP2 UP
OR 80.01  ; HOMEPOST STP2 UP
ANDNOT 11.05  ; MASTER OFF
ANDNOT 60.01  ; FAULT
AND 11.04  ; IR MASTER ON
ANDNOT 3.07  ; RSUP STP2
OUT 3300.07  ; OUT STP2 UP
; rung 39
LD 11.11  ; IR MAN STP2 DN
OR 20.03  ; AUTO STP2 DOWN
OR 90.04  ; ALL STOPPER DOWN
ANDNOT 11.05  ; MASTER OFF
ANDNOT 60.01  ; FAULT
AND 11.04  ; IR MASTER ON
ANDNOT 3.08  ; RSDN STP2
OUT 3300.06  ; OUT STP2 DN
; rung 40
LD 11.12  ; IR MAN STP3 UP
OR 19.08  ; AUTO STP3 UP
OR 80.02  ; HOMEPOST STP3 UP
ANDNOT 11.05  ; MASTER OFF
ANDNOT 60.01  ; FAULT
AND 11.04  ; IR MASTER ON
ANDNOT 3.05  ; RSUP STP3
OUT 3300.09  ; OUT STP3 UP
; rung 41
LD 11.13  ; IR MAN STP3 DN
OR 19.06  ; AUTO STP3 DOWN
OR 90.04  ; ALL STOPPER DOWN
ANDNOT 11.05  ; MASTER OFF
ANDNOT 60.01  ; FAULT
AND 11.04  ; IR MASTER ON
ANDNOT 3.06  ; RSDN STP3
OUT 3300.08  ; OUT STP3 DN
; rung 42
LD 11.14  ; IR MAN STP4 UP
OR 19.03  ; AUTO STP4 UP
OR 80.03  ; HOMEPOST STP4 UP
ANDNOT 11.05  ; MASTER OFF
ANDNOT 60.01  ; FAULT
AND 11.04  ; IR MASTER ON
ANDNOT 3.03  ; RSUP STP4
OUT 3300.11  ; OUT STP4 UP

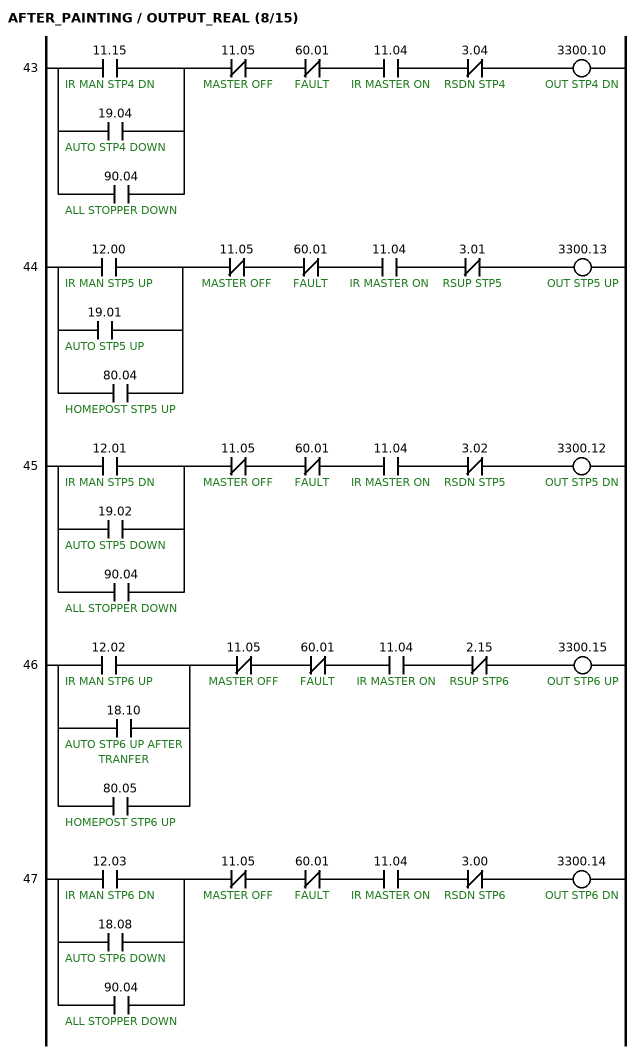
; rung 43
LD 11.15  ; IR MAN STP4 DN
OR 19.04  ; AUTO STP4 DOWN
OR 90.04  ; ALL STOPPER DOWN
ANDNOT 11.05  ; MASTER OFF
ANDNOT 60.01  ; FAULT
AND 11.04  ; IR MASTER ON
ANDNOT 3.04  ; RSDN STP4
OUT 3300.10  ; OUT STP4 DN
; rung 44
LD 12.00  ; IR MAN STP5 UP
OR 19.01  ; AUTO STP5 UP
OR 80.04  ; HOMEPOST STP5 UP
ANDNOT 11.05  ; MASTER OFF
ANDNOT 60.01  ; FAULT
AND 11.04  ; IR MASTER ON
ANDNOT 3.01  ; RSUP STP5
OUT 3300.13  ; OUT STP5 UP
; rung 45
LD 12.01  ; IR MAN STP5 DN
OR 19.02  ; AUTO STP5 DOWN
OR 90.04  ; ALL STOPPER DOWN
ANDNOT 11.05  ; MASTER OFF
ANDNOT 60.01  ; FAULT
AND 11.04  ; IR MASTER ON
ANDNOT 3.02  ; RSDN STP5
OUT 3300.12  ; OUT STP5 DN
; rung 46
LD 12.02  ; IR MAN STP6 UP
OR 18.10  ; AUTO STP6 UP AFTER TRANFER
OR 80.05  ; HOMEPOST STP6 UP
ANDNOT 11.05  ; MASTER OFF
ANDNOT 60.01  ; FAULT
AND 11.04  ; IR MASTER ON
ANDNOT 2.15  ; RSUP STP6
OUT 3300.15  ; OUT STP6 UP
; rung 47
LD 12.03  ; IR MAN STP6 DN
OR 18.08  ; AUTO STP6 DOWN
OR 90.04  ; ALL STOPPER DOWN
ANDNOT 11.05  ; MASTER OFF
ANDNOT 60.01  ; FAULT
AND 11.04  ; IR MASTER ON
ANDNOT 3.00  ; RSDN STP6
OUT 3300.14  ; OUT STP6 DN

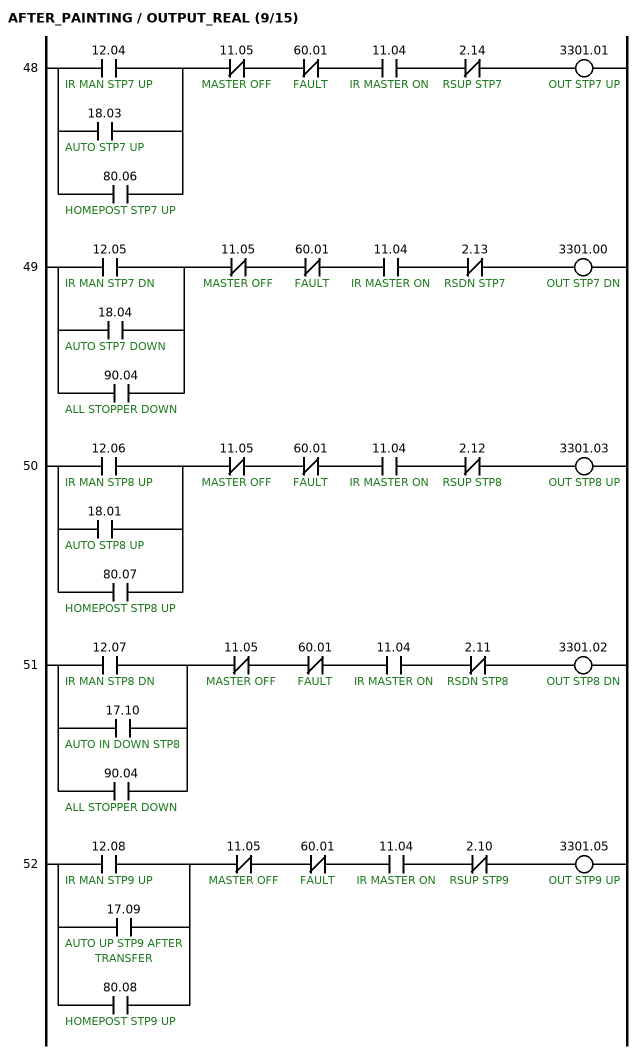
; rung 48
LD 12.04  ; IR MAN STP7 UP
OR 18.03  ; AUTO STP7 UP
OR 80.06  ; HOMEPOST STP7 UP
ANDNOT 11.05  ; MASTER OFF
ANDNOT 60.01  ; FAULT
AND 11.04  ; IR MASTER ON
ANDNOT 2.14  ; RSUP STP7
OUT 3301.01  ; OUT STP7 UP
; rung 49
LD 12.05  ; IR MAN STP7 DN
OR 18.04  ; AUTO STP7 DOWN
OR 90.04  ; ALL STOPPER DOWN
ANDNOT 11.05  ; MASTER OFF
ANDNOT 60.01  ; FAULT
AND 11.04  ; IR MASTER ON
ANDNOT 2.13  ; RSDN STP7
OUT 3301.00  ; OUT STP7 DN
; rung 50
LD 12.06  ; IR MAN STP8 UP
OR 18.01  ; AUTO STP8 UP
OR 80.07  ; HOMEPOST STP8 UP
ANDNOT 11.05  ; MASTER OFF
ANDNOT 60.01  ; FAULT
AND 11.04  ; IR MASTER ON
ANDNOT 2.12  ; RSUP STP8
OUT 3301.03  ; OUT STP8 UP
; rung 51
LD 12.07  ; IR MAN STP8 DN
OR 17.10  ; AUTO IN DOWN STP8
OR 90.04  ; ALL STOPPER DOWN
ANDNOT 11.05  ; MASTER OFF
ANDNOT 60.01  ; FAULT
AND 11.04  ; IR MASTER ON
ANDNOT 2.11  ; RSDN STP8
OUT 3301.02  ; OUT STP8 DN
; rung 52
LD 12.08  ; IR MAN STP9 UP
OR 17.09  ; AUTO UP STP9 AFTER TRANSFER
OR 80.08  ; HOMEPOST STP9 UP
ANDNOT 11.05  ; MASTER OFF
ANDNOT 60.01  ; FAULT
AND 11.04  ; IR MASTER ON
ANDNOT 2.10  ; RSUP STP9
OUT 3301.05  ; OUT STP9 UP

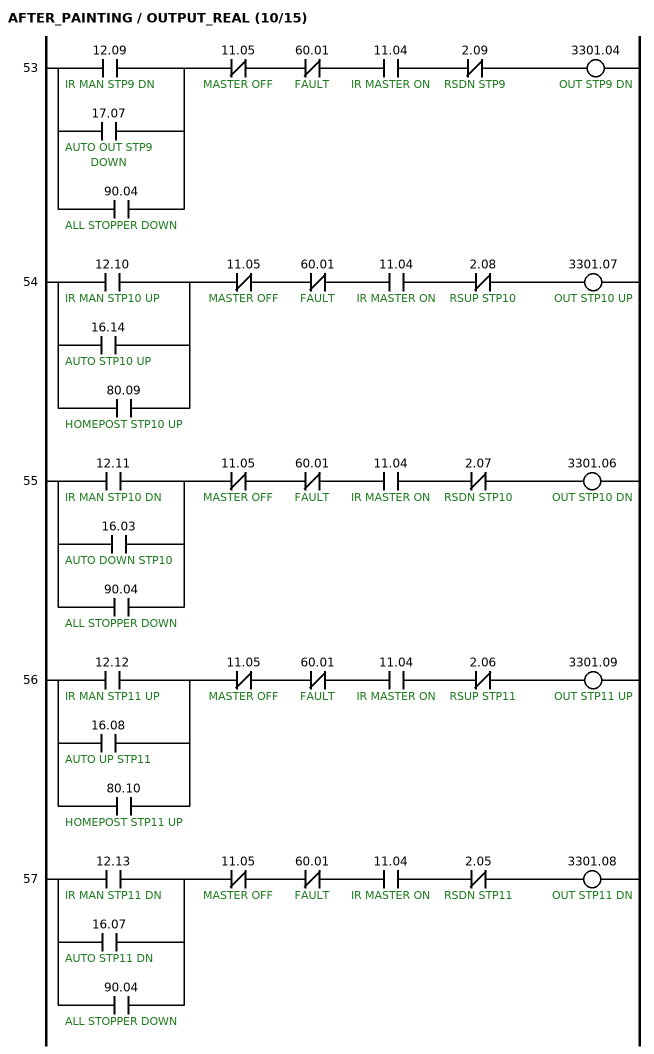
; rung 53
LD 12.09  ; IR MAN STP9 DN
OR 17.07  ; AUTO OUT STP9 DOWN
OR 90.04  ; ALL STOPPER DOWN
ANDNOT 11.05  ; MASTER OFF
ANDNOT 60.01  ; FAULT
AND 11.04  ; IR MASTER ON
ANDNOT 2.09  ; RSDN STP9
OUT 3301.04  ; OUT STP9 DN
; rung 54
LD 12.10  ; IR MAN STP10 UP
OR 16.14  ; AUTO STP10 UP
OR 80.09  ; HOMEPOST STP10 UP
ANDNOT 11.05  ; MASTER OFF
ANDNOT 60.01  ; FAULT
AND 11.04  ; IR MASTER ON
ANDNOT 2.08  ; RSUP STP10
OUT 3301.07  ; OUT STP10 UP
; rung 55
LD 12.11  ; IR MAN STP10 DN
OR 16.03  ; AUTO DOWN STP10
OR 90.04  ; ALL STOPPER DOWN
ANDNOT 11.05  ; MASTER OFF
ANDNOT 60.01  ; FAULT
AND 11.04  ; IR MASTER ON
ANDNOT 2.07  ; RSDN STP10
OUT 3301.06  ; OUT STP10 DN
; rung 56
LD 12.12  ; IR MAN STP11 UP
OR 16.08  ; AUTO UP STP11
OR 80.10  ; HOMEPOST STP11 UP
ANDNOT 11.05  ; MASTER OFF
ANDNOT 60.01  ; FAULT
AND 11.04  ; IR MASTER ON
ANDNOT 2.06  ; RSUP STP11
OUT 3301.09  ; OUT STP11 UP
; rung 57
LD 12.13  ; IR MAN STP11 DN
OR 16.07  ; AUTO STP11 DN
OR 90.04  ; ALL STOPPER DOWN
ANDNOT 11.05  ; MASTER OFF
ANDNOT 60.01  ; FAULT
AND 11.04  ; IR MASTER ON
ANDNOT 2.05  ; RSDN STP11
OUT 3301.08  ; OUT STP11 DN

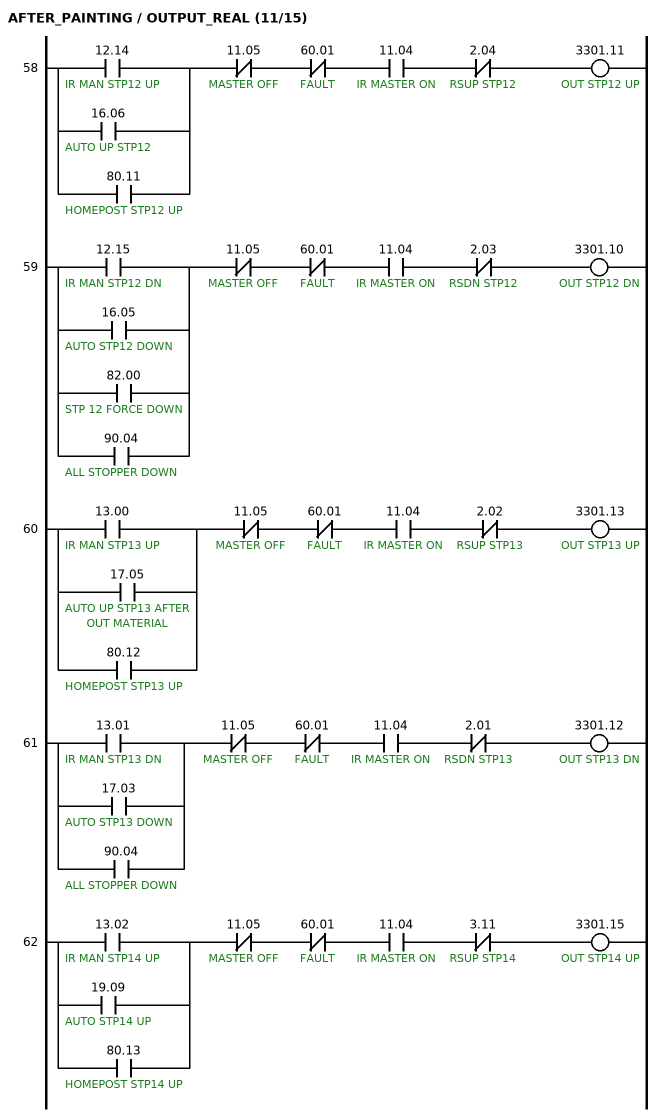
; rung 58
LD 12.14  ; IR MAN STP12 UP
OR 16.06  ; AUTO UP STP12
OR 80.11  ; HOMEPOST STP12 UP
ANDNOT 11.05  ; MASTER OFF
ANDNOT 60.01  ; FAULT
AND 11.04  ; IR MASTER ON
ANDNOT 2.04  ; RSUP STP12
OUT 3301.11  ; OUT STP12 UP
; rung 59
LD 12.15  ; IR MAN STP12 DN
OR 16.05  ; AUTO STP12 DOWN
OR 82.00  ; STP 12 FORCE DOWN
OR 90.04  ; ALL STOPPER DOWN
ANDNOT 11.05  ; MASTER OFF
ANDNOT 60.01  ; FAULT
AND 11.04  ; IR MASTER ON
ANDNOT 2.03  ; RSDN STP12
OUT 3301.10  ; OUT STP12 DN
; rung 60
LD 13.00  ; IR MAN STP13 UP
OR 17.05  ; AUTO UP STP13 AFTER OUT MATERIAL
OR 80.12  ; HOMEPOST STP13 UP
ANDNOT 11.05  ; MASTER OFF
ANDNOT 60.01  ; FAULT
AND 11.04  ; IR MASTER ON
ANDNOT 2.02  ; RSUP STP13
OUT 3301.13  ; OUT STP13 UP
; rung 61
LD 13.01  ; IR MAN STP13 DN
OR 17.03  ; AUTO STP13 DOWN
OR 90.04  ; ALL STOPPER DOWN
ANDNOT 11.05  ; MASTER OFF
ANDNOT 60.01  ; FAULT
AND 11.04  ; IR MASTER ON
ANDNOT 2.01  ; RSDN STP13
OUT 3301.12  ; OUT STP13 DN
; rung 62
LD 13.02  ; IR MAN STP14 UP
OR 19.09  ; AUTO STP14 UP
OR 80.13  ; HOMEPOST STP14 UP
ANDNOT 11.05  ; MASTER OFF
ANDNOT 60.01  ; FAULT
AND 11.04  ; IR MASTER ON
ANDNOT 3.11  ; RSUP STP14
OUT 3301.15  ; OUT STP14 UP

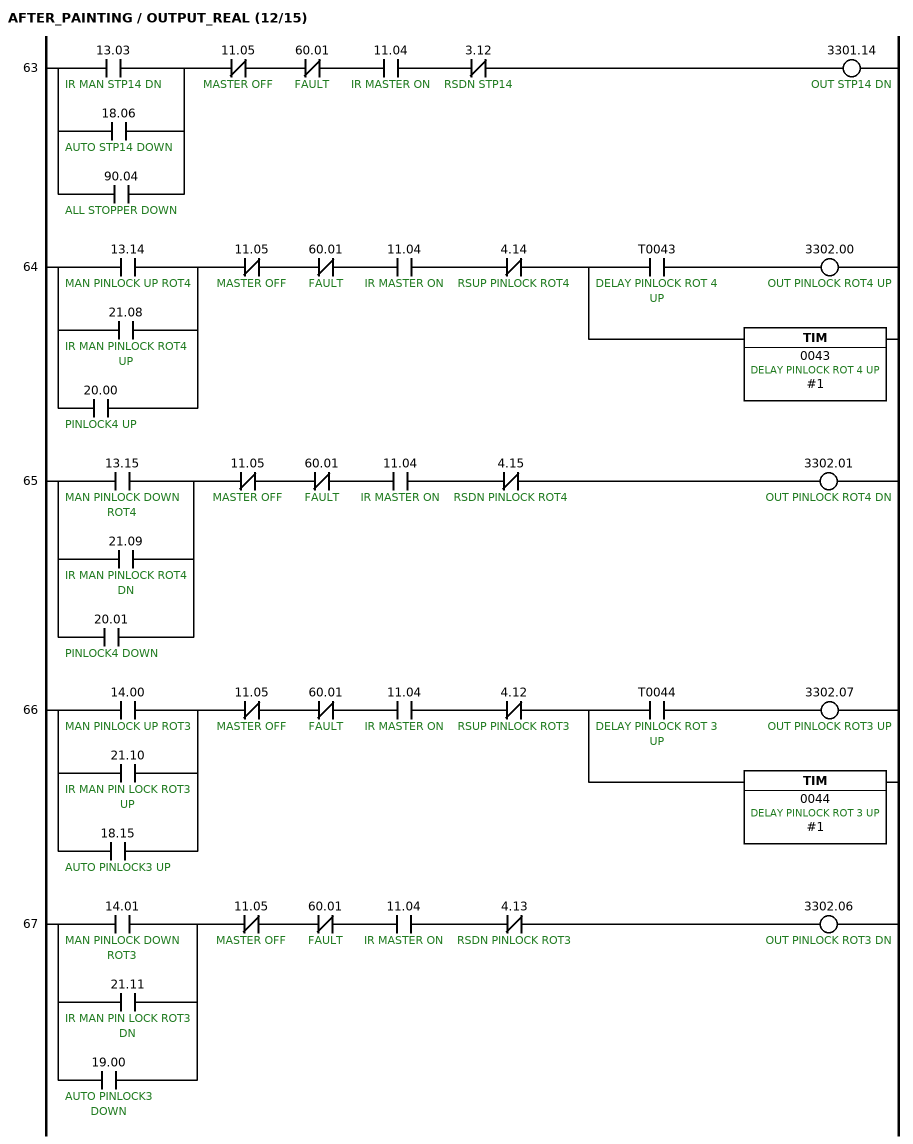
; rung 63
LD 13.03  ; IR MAN STP14 DN
OR 18.06  ; AUTO STP14 DOWN
OR 90.04  ; ALL STOPPER DOWN
ANDNOT 11.05  ; MASTER OFF
ANDNOT 60.01  ; FAULT
AND 11.04  ; IR MASTER ON
ANDNOT 3.12  ; RSDN STP14
OUT 3301.14  ; OUT STP14 DN
; rung 64
LD 13.14  ; MAN PINLOCK UP ROT4
OR 21.08  ; IR MAN PINLOCK ROT4 UP
OR 20.00  ; PINLOCK4 UP
ANDNOT 11.05  ; MASTER OFF
ANDNOT 60.01  ; FAULT
AND 11.04  ; IR MASTER ON
ANDNOT 4.14  ; RSUP PINLOCK ROT4
OUT TR0
AND T0043  ; DELAY PINLOCK ROT 4 UP
OUT 3302.00  ; OUT PINLOCK ROT4 UP
LD TR0
TIM 0043 #1  ; DELAY PINLOCK ROT 4 UP
; rung 65
LD 13.15  ; MAN PINLOCK DOWN ROT4
OR 21.09  ; IR MAN PINLOCK ROT4 DN
OR 20.01  ; PINLOCK4 DOWN
ANDNOT 11.05  ; MASTER OFF
ANDNOT 60.01  ; FAULT
AND 11.04  ; IR MASTER ON
ANDNOT 4.15  ; RSDN PINLOCK ROT4
OUT 3302.01  ; OUT PINLOCK ROT4 DN
; rung 66
LD 14.00  ; MAN PINLOCK UP ROT3
OR 21.10  ; IR MAN PIN LOCK ROT3 UP
OR 18.15  ; AUTO PINLOCK3 UP
ANDNOT 11.05  ; MASTER OFF
ANDNOT 60.01  ; FAULT
AND 11.04  ; IR MASTER ON
ANDNOT 4.12  ; RSUP PINLOCK ROT3
OUT TR0
AND T0044  ; DELAY PINLOCK ROT 3 UP
OUT 3302.07  ; OUT PINLOCK ROT3 UP
LD TR0
TIM 0044 #1  ; DELAY PINLOCK ROT 3 UP
; rung 67
LD 14.01  ; MAN PINLOCK DOWN ROT3
OR 21.11  ; IR MAN PIN LOCK ROT3 DN
OR 19.00  ; AUTO PINLOCK3 DOWN
ANDNOT 11.05  ; MASTER OFF
ANDNOT 60.01  ; FAULT
AND 11.04  ; IR MASTER ON
ANDNOT 4.13  ; RSDN PINLOCK ROT3
OUT 3302.06  ; OUT PINLOCK ROT3 DN

